KUKA KRL program: MyProgram_026().src

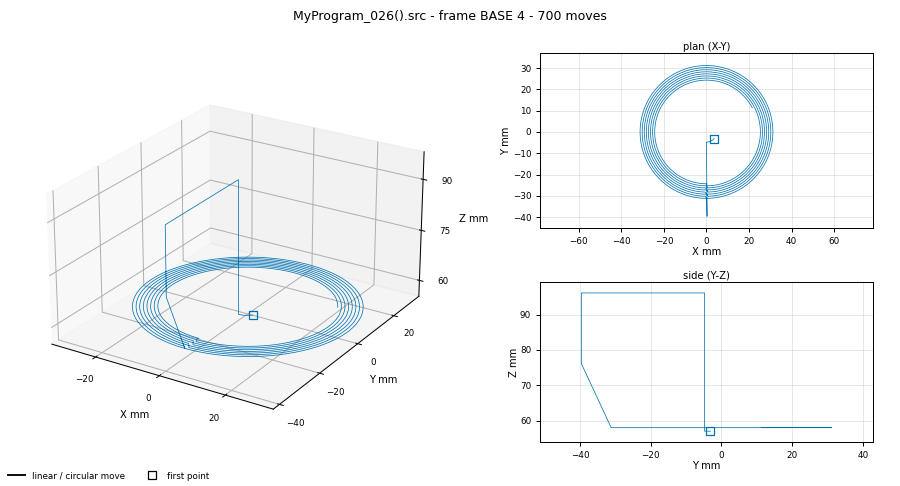
[picture p0: tool path of MyProgram_026().src in frame BASE 4, 700 of 700 moves have a stored position in this frame; points joined in program order, loops and branches not executed]
&ACCESS RVP
&REL 1
&PARAM TEMPLATE = C:\KRC\Roboter\Template\vorgabe
&PARAM EDITMASK = *
DEF MyProgram_026()
; ---- Setting reference (Base) ----
$BASE = BASE_DATA[4]

; --------------------------
; ---- Setting tool (TCP) ----
$TOOL = TOOL_DATA[3]
; --------------------------

$VEL.CP = VEL_APROX_PRINT
Startdeposition()
$VEL.CP = VEL_PRINT
LIN {X 3.5971,Y -3.1129,Z 57,A -2.6409,B 0,C 0,E1 0.1598,E2 -629.9281} C_DIS
LIN {X 2.9999,Y -3.6921,Z 57,A -2.6876,B 0,C 0,E1 0.1598,E2 -629.9281} C_DIS
LIN {X 2.3555,Y -4.1313,Z 57,A -2.7301,B 0,C 0,E1 0.1598,E2 -629.9281} C_DIS
LIN {X 1.6977,Y -4.4434,Z 57,A -2.7676,B 0,C 0,E1 0.1598,E2 -629.9281} C_DIS
LIN {X 0.8464,Y -4.6808,Z 57,A -2.809,B 0,C 0,E1 0.1598,E2 -629.9281} C_DIS
LIN {X -0.0081,Y -4.7574,Z 57,A -2.8436,B 0,C 0,E1 0.1598,E2 -629.9282} C_DIS
Enddeposition()
LIN {X -0.0081,Y -4.7574,Z 62,A -2.8335,B 0,C 0,E1 0.1598,E2 -629.928} C_DIS
LIN {X -0.0081,Y -4.7573,Z 77,A -2.8076,B 0,C 0,E1 0.1598,E2 -629.9269} C_DIS
LIN {X -0.0081,Y -4.7573,Z 96.1262,A -2.7825,B 0,C 0,E1 0.1598,E2 -629.9267} C_DIS
LIN {X 0.2603,Y -39.6445,Z 96.1262,A -95.8861,B 24.839,C -2.9274,E1 25.0032,E2 -541.4173} C_DIS
LIN {X 0.2603,Y -39.6445,Z 76.1262,A -95.5567,B 24.8539,C -2.789,E1 25.0032,E2 -541.4173} C_DIS
LIN {X 0.1436,Y -33.3063,Z 62.5315,A -95.5942,B 24.8522,C -2.8048,E1 25.0032,E2 -541.4173} C_DIS
LIN {X 0.1047,Y -31.1935,Z 58,A -95.6082,B 24.8516,C -2.8106,E1 25.0032,E2 -541.4173} C_DIS
Startdeposition()
$VEL.CP = VEL_PRINT
LIN {X 2.2949,Y -31.1109,Z 58,A -91.3981,B 24.8512,C -2.8143,E1 25.015,E2 -545.6344} C_DIS
LIN {X 4.5773,Y -30.8578,Z 58,A -87.1855,B 24.8509,C -2.8169,E1 25.0267,E2 -549.8498} C_DIS
LIN {X 6.835,Y -30.4375,Z 58,A -82.975,B 24.8506,C -2.8204,E1 25.0382,E2 -554.0634} C_DIS
LIN {X 9.0556,Y -29.8522,Z 58,A -78.7668,B 24.8501,C -2.8248,E1 25.0495,E2 -558.275} C_DIS
LIN {X 11.2271,Y -29.1051,Z 58,A -74.5606,B 24.8495,C -2.83,E1 25.0606,E2 -562.485} C_DIS
LIN {X 13.3378,Y -28.2004,Z 58,A -70.3565,B 24.8489,C -2.8362,E1 25.0713,E2 -566.6932} C_DIS
LIN {X 15.3762,Y -27.1428,Z 58,A -66.1541,B 24.8481,C -2.8431,E1 25.0816,E2 -570.8999} C_DIS
LIN {X 17.3313,Y -25.9381,Z 58,A -61.9537,B 24.8473,C -2.8508,E1 25.0915,E2 -575.1049} C_DIS
LIN {X 19.1924,Y -24.5928,Z 58,A -57.755,B 24.8464,C -2.8592,E1 25.1008,E2 -579.3084} C_DIS
LIN {X 20.9496,Y -23.1143,Z 58,A -53.558,B 24.8454,C -2.8683,E1 25.1097,E2 -583.5105} C_DIS
LIN {X 22.5932,Y -21.5105,Z 58,A -49.3625,B 24.8444,C -2.8781,E1 25.1179,E2 -587.7112} C_DIS
LIN {X 24.1144,Y -19.7902,Z 58,A -45.1683,B 24.8432,C -2.8884,E1 25.1255,E2 -591.9108} C_DIS
LIN {X 25.5049,Y -17.9626,Z 58,A -40.9754,B 24.8421,C -2.8993,E1 25.1324,E2 -596.1092} C_DIS
LIN {X 26.7572,Y -16.0377,Z 58,A -36.7836,B 24.8408,C -2.9106,E1 25.1386,E2 -600.3066} C_DIS
LIN {X 27.8645,Y -14.0258,Z 58,A -32.5927,B 24.8395,C -2.9223,E1 25.1441,E2 -604.5031} C_DIS
LIN {X 28.8208,Y -11.938,Z 58,A -28.4027,B 24.8382,C -2.9344,E1 25.1488,E2 -608.6988} C_DIS
LIN {X 29.621,Y -9.7854,Z 58,A -24.2134,B 24.8368,C -2.9467,E1 25.1527,E2 -612.8938} C_DIS
LIN {X 30.2606,Y -7.5799,Z 58,A -20.0245,B 24.8354,C -2.9593,E1 25.1557,E2 -617.0884} C_DIS
LIN {X 30.7362,Y -5.3332,Z 58,A -15.836,B 24.834,C -2.972,E1 25.1579,E2 -621.2824} C_DIS
LIN {X 31.0452,Y -3.0577,Z 58,A -11.6476,B 24.8326,C -2.9848,E1 25.1593,E2 -625.4764} C_DIS
LIN {X 31.1861,Y -0.7656,Z 58,A -8.1402,B 24.8322,C -2.9882,E1 25.1598,E2 -628.9711} C_DIS
LIN {X 31.1915,Y 0.4681,Z 58,A -5.3067,B 24.8305,C -3.0031,E1 25.1597,E2 -631.8229} C_DIS
LIN {X 31.0804,Y 2.6765,Z 58,A -1.1766,B 24.829,C -3.0166,E1 25.1589,E2 -635.9605} C_DIS
LIN {X 30.7993,Y 4.9557,Z 58,A 3.0123,B 24.8275,C -3.0291,E1 25.1573,E2 -640.1544} C_DIS
LIN {X 30.3513,Y 7.208,Z 58,A 7.2019,B 24.8261,C -3.0414,E1 25.1548,E2 -644.3487} C_DIS
LIN {X 29.7388,Y 9.4212,Z 58,A 11.392,B 24.8247,C -3.0534,E1 25.1514,E2 -648.5433} C_DIS
LIN {X 28.9652,Y 11.5834,Z 58,A 15.583,B 24.8234,C -3.065,E1 25.1473,E2 -652.7386} C_DIS
LIN {X 28.0346,Y 13.6828,Z 58,A 19.7751,B 24.8221,C -3.0763,E1 25.1423,E2 -656.9345} C_DIS
LIN {X 26.952,Y 15.7081,Z 58,A 23.9682,B 24.8208,C -3.087,E1 25.1366,E2 -661.1313} C_DIS
LIN {X 25.7234,Y 17.6483,Z 58,A 28.1627,B 24.8197,C -3.0972,E1 25.1301,E2 -665.3291} C_DIS
LIN {X 24.3555,Y 19.4928,Z 58,A 32.3584,B 24.8185,C -3.1068,E1 25.123,E2 -669.5278} C_DIS
LIN {X 22.8555,Y 21.2317,Z 58,A 36.5559,B 24.8175,C -3.1158,E1 25.1152,E2 -673.7278} C_DIS
LIN {X 21.2317,Y 22.8555,Z 58,A 40.7549,B 24.8165,C -3.1241,E1 25.1067,E2 -677.929} C_DIS
LIN {X 19.4928,Y 24.3555,Z 58,A 44.9555,B 24.8156,C -3.1316,E1 25.0977,E2 -682.1315} C_DIS
LIN {X 17.6483,Y 25.7234,Z 58,A 49.1582,B 24.8148,C -3.1384,E1 25.0881,E2 -686.3356} C_DIS
LIN {X 15.7081,Y 26.952,Z 58,A 53.3628,B 24.8141,C -3.1444,E1 25.0781,E2 -690.5412} C_DIS
LIN {X 13.6828,Y 28.0346,Z 58,A 57.5693,B 24.8135,C -3.1495,E1 25.0676,E2 -694.7483} C_DIS
LIN {X 11.5834,Y 28.9652,Z 58,A 61.7781,B 24.813,C -3.1537,E1 25.0568,E2 -698.9572} C_DIS
LIN {X 9.4212,Y 29.7388,Z 58,A 65.9888,B 24.8126,C -3.157,E1 25.0457,E2 -703.1677} C_DIS
LIN {X 7.208,Y 30.3513,Z 58,A 70.2017,B 24.8123,C -3.1595,E1 25.0343,E2 -707.38} C_DIS
LIN {X 4.9557,Y 30.7993,Z 58,A 74.4171,B 24.8121,C -3.161,E1 25.0227,E2 -711.5942} C_DIS
LIN {X 2.6765,Y 31.0804,Z 58,A 78.6345,B 24.8121,C -3.1615,E1 25.011,E2 -715.8102} C_DIS
LIN {X 0.3828,Y 31.1931,Z 58,A 82.8541,B 24.8121,C -3.1611,E1 24.9992,E2 -720.028} C_DIS
LIN {X -1.9129,Y 31.1367,Z 58,A 87.0743,B 24.8123,C -3.1597,E1 24.9875,E2 -724.2458} C_DIS
LIN {X -4.1983,Y 30.9117,Z 58,A 91.3003,B 24.8125,C -3.1575,E1 24.9757,E2 -728.4692} C_DIS
LIN {X -6.4609,Y 30.5191,Z 58,A 95.5267,B 24.8129,C -3.1543,E1 24.9642,E2 -732.6926} C_DIS
LIN {X -8.6885,Y 29.9611,Z 58,A 99.7553,B 24.8134,C -3.1501,E1 24.9528,E2 -736.9178} C_DIS
LIN {X -10.8691,Y 29.2407,Z 58,A 103.9859,B 24.814,C -3.1451,E1 24.9416,E2 -741.1448} C_DIS
LIN {X -12.9907,Y 28.3619,Z 58,A 108.2187,B 24.8147,C -3.1393,E1 24.9308,E2 -745.3735} C_DIS
LIN {X -15.0419,Y 27.3294,Z 58,A 112.4534,B 24.8155,C -3.1326,E1 24.9204,E2 -749.6039} C_DIS
LIN {X -17.0117,Y 26.1488,Z 58,A 116.6901,B 24.8164,C -3.1251,E1 24.9104,E2 -753.836} C_DIS
LIN {X -18.8892,Y 24.8265,Z 58,A 120.9285,B 24.8174,C -3.1168,E1 24.9008,E2 -758.0696} C_DIS
LIN {X -20.6644,Y 23.3697,Z 58,A 125.1687,B 24.8184,C -3.1078,E1 24.8918,E2 -762.3048} C_DIS
LIN {X -22.3275,Y 21.7862,Z 58,A 129.4103,B 24.8195,C -3.0982,E1 24.8834,E2 -766.5412} C_DIS
LIN {X -23.8697,Y 20.0846,Z 58,A 133.6535,B 24.8207,C -3.0879,E1 24.8756,E2 -770.779} C_DIS
LIN {X -25.2826,Y 18.2742,Z 58,A 137.8979,B 24.822,C -3.0771,E1 24.8685,E2 -775.018} C_DIS
LIN {X -26.5584,Y 16.3648,Z 58,A 142.1437,B 24.8233,C -3.0658,E1 24.8621,E2 -779.2582} C_DIS
LIN {X -27.6903,Y 14.3667,Z 58,A 146.3904,B 24.8247,C -3.0541,E1 24.8565,E2 -783.4992} C_DIS
LIN {X -28.6722,Y 12.2908,Z 58,A 150.638,B 24.8261,C -3.042,E1 24.8516,E2 -787.7411} C_DIS
LIN {X -29.4987,Y 10.1482,Z 58,A 154.8864,B 24.8275,C -3.0296,E1 24.8476,E2 -791.9838} C_DIS
LIN {X -30.1653,Y 7.9506,Z 58,A 159.1351,B 24.8289,C -3.0169,E1 24.8443,E2 -796.2268} C_DIS
LIN {X -30.6684,Y 5.71,Z 58,A 163.3845,B 24.8304,C -3.0041,E1 24.842,E2 -800.4706} C_DIS
LIN {X -31.0054,Y 3.4384,Z 58,A 167.634,B 24.8318,C -2.9912,E1 24.8405,E2 -804.7145} C_DIS
LIN {X -31.1743,Y 1.1482,Z 58,A 171.597,B 24.8335,C -2.9761,E1 24.8398,E2 -808.6653} C_DIS
LIN {X -31.1861,Y -0.7656,Z 58,A 175.4249,B 24.8345,C -2.9675,E1 24.8399,E2 -812.4955} C_DIS
LIN {X -31.0452,Y -3.0577,Z 58,A 179.674,B 24.8359,C -2.9547,E1 24.8409,E2 -816.7395} C_DIS
LIN {X -30.7362,Y -5.3332,Z 58,A -176.0771,B 24.8373,C -2.942,E1 24.8427,E2 -820.9834} C_DIS
LIN {X -30.2606,Y -7.5799,Z 58,A -171.8289,B 24.8387,C -2.9296,E1 24.8454,E2 -825.2269} C_DIS
LIN {X -29.621,Y -9.7854,Z 58,A -167.5814,B 24.84,C -2.9176,E1 24.8489,E2 -829.4699} C_DIS
LIN {X -28.8208,Y -11.938,Z 58,A -163.3348,B 24.8413,C -2.9059,E1 24.8532,E2 -833.7123} C_DIS
LIN {X -27.8645,Y -14.0258,Z 58,A -159.0893,B 24.8426,C -2.8946,E1 24.8583,E2 -837.954} C_DIS
LIN {X -26.7572,Y -16.0377,Z 58,A -154.845,B 24.8437,C -2.8839,E1 24.8642,E2 -842.1947} C_DIS
LIN {X -25.5049,Y -17.9626,Z 58,A -150.602,B 24.8448,C -2.8737,E1 24.8709,E2 -846.4344} C_DIS
LIN {X -24.1144,Y -19.7902,Z 58,A -146.3605,B 24.8459,C -2.8641,E1 24.8782,E2 -850.673} C_DIS
LIN {X -22.5932,Y -21.5105,Z 58,A -142.1207,B 24.8468,C -2.8553,E1 24.8862,E2 -854.9103} C_DIS
LIN {X -20.9496,Y -23.1143,Z 58,A -137.8825,B 24.8477,C -2.8471,E1 24.8948,E2 -859.1464} C_DIS
LIN {X -19.1924,Y -24.5928,Z 58,A -133.6461,B 24.8485,C -2.8397,E1 24.904,E2 -863.381} C_DIS
LIN {X -17.3313,Y -25.9381,Z 58,A -129.4116,B 24.8492,C -2.8331,E1 24.9137,E2 -867.6141} C_DIS
LIN {X -15.3762,Y -27.1428,Z 58,A -125.1792,B 24.8498,C -2.8274,E1 24.9239,E2 -871.8456} C_DIS
LIN {X -13.3378,Y -28.2004,Z 58,A -120.9489,B 24.8503,C -2.8225,E1 24.9345,E2 -876.0755} C_DIS
LIN {X -11.2271,Y -29.1051,Z 58,A -116.7206,B 24.8508,C -2.8185,E1 24.9454,E2 -880.3037} C_DIS
LIN {X -9.0556,Y -29.8522,Z 58,A -112.4946,B 24.8511,C -2.8154,E1 24.9567,E2 -884.53} C_DIS
LIN {X -6.835,Y -30.4375,Z 58,A -108.2707,B 24.8513,C -2.8133,E1 24.9681,E2 -888.7546} C_DIS
LIN {X -4.5773,Y -30.8578,Z 58,A -104.0493,B 24.8514,C -2.8121,E1 24.9797,E2 -892.9773} C_DIS
LIN {X -2.2949,Y -31.1109,Z 58,A -99.8299,B 24.8514,C -2.8119,E1 24.9915,E2 -897.1982} C_DIS
LIN {X 0.1047,Y -31.1935,Z 58,A -95.6081,B 24.8516,C -2.8106,E1 25.0033,E2 -901.4173} C_DIS
Enddeposition()
LIN {X 0.1047,Y -31.1935,Z 58,A -95.6081,B 24.8516,C -2.8106,E1 25.0033,E2 -901.4173} C_DIS
Startdeposition()
$VEL.CP = VEL_PRINT
LIN {X -0.5457,Y -30.2108,Z 58,A -98.6907,B 24.8519,C -2.8079,E1 24.9946,E2 -898.3283} C_DIS
LIN {X -2.6136,Y -30.1028,Z 58,A -102.6666,B 24.8519,C -2.8074,E1 24.9835,E2 -894.3496} C_DIS
LIN {X -4.817,Y -29.8297,Z 58,A -106.8223,B 24.8518,C -2.8088,E1 24.9721,E2 -890.194} C_DIS
LIN {X -6.6677,Y -29.4712,Z 58,A -110.3863,B 24.8516,C -2.8104,E1 24.9623,E2 -886.6296} C_DIS
LIN {X -9.1107,Y -28.8099,Z 58,A -115.271,B 24.8514,C -2.8128,E1 24.9492,E2 -881.7424} C_DIS
LIN {X -11.2355,Y -28.0496,Z 58,A -119.5455,B 24.851,C -2.8166,E1 24.9381,E2 -877.4682} C_DIS
LIN {X -13.2679,Y -27.1474,Z 58,A -123.8987,B 24.8506,C -2.8202,E1 24.927,E2 -873.1125} C_DIS
LIN {X -15.1376,Y -26.1506,Z 58,A -127.6644,B 24.8498,C -2.8276,E1 24.9179,E2 -869.3537} C_DIS
LIN {X -16.7352,Y -25.1583,Z 58,A -131.3179,B 24.8493,C -2.8322,E1 24.9093,E2 -865.6995} C_DIS
LIN {X -18.2715,Y -24.0658,Z 58,A -134.908,B 24.8487,C -2.8381,E1 24.9012,E2 -862.1106} C_DIS
LIN {X -19.7968,Y -22.8273,Z 58,A -138.5955,B 24.8479,C -2.8452,E1 24.8933,E2 -858.4261} C_DIS
LIN {X -21.2071,Y -21.5232,Z 58,A -142.6762,B 24.8475,C -2.8491,E1 24.8851,E2 -854.3376} C_DIS
LIN {X -22.8019,Y -19.8259,Z 58,A -147.2693,B 24.8466,C -2.8574,E1 24.8766,E2 -849.7438} C_DIS
LIN {X -24.601,Y -17.5437,Z 58,A -152.3405,B 24.8448,C -2.8737,E1 24.8681,E2 -844.6872} C_DIS
LIN {X -25.8525,Y -15.6411,Z 58,A -156.1895,B 24.8433,C -2.888,E1 24.8623,E2 -840.853} C_DIS
LIN {X -26.6221,Y -14.2922,Z 58,A -159.6438,B 24.8429,C -2.892,E1 24.8576,E2 -837.3901} C_DIS
LIN {X -27.5197,Y -12.4764,Z 58,A -163.3944,B 24.8416,C -2.9031,E1 24.8531,E2 -833.6458} C_DIS
LIN {X -28.3033,Y -10.5797,Z 58,A -167.0641,B 24.8403,C -2.9156,E1 24.8494,E2 -829.9855} C_DIS
LIN {X -28.8908,Y -8.85,Z 58,A -171.2263,B 24.8397,C -2.9208,E1 24.8458,E2 -825.812} C_DIS
LIN {X -29.507,Y -6.506,Z 58,A -175.4387,B 24.8379,C -2.9372,E1 24.843,E2 -821.614} C_DIS
LIN {X -29.8601,Y -4.6221,Z 58,A -179.4869,B 24.837,C -2.9454,E1 24.8412,E2 -817.5615} C_DIS
LIN {X -30.0965,Y -2.6829,Z 58,A 177.5499,B 24.8351,C -2.9618,E1 24.8403,E2 -814.6198} C_DIS
LIN {X -30.1951,Y -1.1291,Z 58,A 174.0998,B 24.8345,C -2.9676,E1 24.8398,E2 -811.1628} C_DIS
LIN {X -30.2137,Y 0.3884,Z 58,A 171.1347,B 24.8335,C -2.976,E1 24.8398,E2 -808.2} C_DIS
LIN {X -30.0111,Y 3.506,Z 58,A 164.6989,B 24.8318,C -2.9911,E1 24.8414,E2 -801.7618} C_DIS
LIN {X -29.5072,Y 6.5047,Z 58,A 158.887,B 24.8299,C -3.0087,E1 24.8445,E2 -795.9576} C_DIS
LIN {X -28.8455,Y 8.9959,Z 58,A 154.669,B 24.8276,C -3.0281,E1 24.8478,E2 -791.7616} C_DIS
LIN {X -28.2324,Y 10.7669,Z 58,A 150.9243,B 24.8266,C -3.0375,E1 24.8513,E2 -788.0182} C_DIS
LIN {X -27.3464,Y 12.852,Z 58,A 146.3112,B 24.8254,C -3.0479,E1 24.8566,E2 -783.4046} C_DIS
LIN {X -25.9429,Y 15.491,Z 58,A 140.9017,B 24.8233,C -3.0656,E1 24.8639,E2 -778.0093} C_DIS
LIN {X -24.8443,Y 17.1975,Z 58,A 137.0408,B 24.8221,C -3.0759,E1 24.8699,E2 -774.1538} C_DIS
LIN {X -23.5808,Y 18.8935,Z 58,A 132.9127,B 24.821,C -3.0855,E1 24.877,E2 -770.0289} C_DIS
LIN {X -22.0567,Y 20.6518,Z 58,A 128.4632,B 24.8198,C -3.096,E1 24.8853,E2 -765.5849} C_DIS
LIN {X -20.8476,Y 21.8722,Z 58,A 125.6303,B 24.8185,C -3.1067,E1 24.8909,E2 -762.7657} C_DIS
LIN {X -19.1986,Y 23.3329,Z 58,A 121.0011,B 24.8179,C -3.1124,E1 24.9007,E2 -758.132} C_DIS
LIN {X -17.428,Y 24.6835,Z 58,A 116.7503,B 24.8169,C -3.1206,E1 24.9102,E2 -753.8859} C_DIS
LIN {X -15.6312,Y 25.8585,Z 58,A 112.7849,B 24.8159,C -3.1289,E1 24.9196,E2 -749.9277} C_DIS
LIN {X -13.8263,Y 26.8669,Z 58,A 109.5725,B 24.8145,C -3.1412,E1 24.9274,E2 -746.7355} C_DIS
LIN {X -12.1506,Y 27.6651,Z 58,A 104.5873,B 24.8153,C -3.1342,E1 24.9401,E2 -741.7214} C_DIS
LIN {X -9.6521,Y 28.6326,Z 58,A 100.3116,B 24.8137,C -3.1474,E1 24.9513,E2 -737.4684} C_DIS
LIN {X -7.4806,Y 29.2751,Z 58,A 95.3533,B 24.8139,C -3.1459,E1 24.9647,E2 -732.499} C_DIS
LIN {X -4.8516,Y 29.824,Z 58,A 90.8217,B 24.8128,C -3.1548,E1 24.9771,E2 -727.9839} C_DIS
LIN {X -2.895,Y 30.0769,Z 58,A 87.058,B 24.8126,C -3.1566,E1 24.9875,E2 -724.2221} C_DIS
LIN {X -0.8345,Y 30.2043,Z 58,A 83.1681,B 24.8124,C -3.1582,E1 24.9984,E2 -720.3349} C_DIS
LIN {X 1.0968,Y 30.1963,Z 58,A 79.3527,B 24.8126,C -3.1572,E1 25.009,E2 -716.5178} C_DIS
LIN {X 2.9201,Y 30.0746,Z 58,A 76.1368,B 24.8123,C -3.1594,E1 25.0179,E2 -713.3089} C_DIS
LIN {X 4.4982,Y 29.8786,Z 58,A 73.3207,B 24.8121,C -3.1607,E1 25.0257,E2 -710.4984} C_DIS
LIN {X 6.1892,Y 29.5752,Z 58,A 69.76,B 24.8127,C -3.1563,E1 25.0355,E2 -706.9313} C_DIS
LIN {X 8.1432,Y 29.0979,Z 58,A 65.9758,B 24.8129,C -3.1543,E1 25.0457,E2 -703.1483} C_DIS
LIN {X 10.3307,Y 28.3948,Z 58,A 61.382,B 24.8136,C -3.1482,E1 25.0579,E2 -698.549} C_DIS
LIN {X 12.0292,Y 27.718,Z 58,A 57.7365,B 24.8143,C -3.1427,E1 25.0673,E2 -694.899} C_DIS
LIN {X 14.7973,Y 26.3445,Z 58,A 52.3919,B 24.8145,C -3.141,E1 25.0805,E2 -689.5652} C_DIS
LIN {X 16.4389,Y 25.3529,Z 58,A 48.6582,B 24.8153,C -3.1345,E1 25.0893,E2 -685.828} C_DIS
LIN {X 17.6927,Y 24.4946,Z 58,A 46.1986,B 24.8153,C -3.1346,E1 25.0949,E2 -683.3773} C_DIS
LIN {X 19.3952,Y 23.1695,Z 58,A 41.6642,B 24.8167,C -3.1221,E1 25.1048,E2 -678.8302} C_DIS
LIN {X 20.9276,Y 21.7951,Z 58,A 37.7631,B 24.8176,C -3.1145,E1 25.1128,E2 -674.9267} C_DIS
LIN {X 22.3953,Y 20.2847,Z 58,A 33.7242,B 24.8187,C -3.1054,E1 25.1205,E2 -670.8838} C_DIS
LIN {X 23.411,Y 19.103,Z 58,A 30.8393,B 24.8194,C -3.0995,E1 25.1257,E2 -667.9983} C_DIS
LIN {X 24.5993,Y 17.5459,Z 58,A 27.1691,B 24.8204,C -3.0912,E1 25.1318,E2 -664.326} C_DIS
LIN {X 25.7265,Y 15.8484,Z 58,A 23.3683,B 24.8214,C -3.0822,E1 25.1375,E2 -660.5231} C_DIS
LIN {X 26.864,Y 13.832,Z 58,A 19.7293,B 24.8216,C -3.0801,E1 25.1424,E2 -656.8981} C_DIS
LIN {X 27.5705,Y 12.3637,Z 58,A 15.7043,B 24.824,C -3.0598,E1 25.1472,E2 -652.8466} C_DIS
LIN {X 28.4448,Y 10.1938,Z 58,A 11.413,B 24.8252,C -3.049,E1 25.1514,E2 -648.5537} C_DIS
LIN {X 29.1291,Y 8.0317,Z 58,A 7.1909,B 24.8266,C -3.0374,E1 25.1548,E2 -644.3282} C_DIS
LIN {X 29.6149,Y 5.9961,Z 58,A 3.4136,B 24.8277,C -3.0279,E1 25.1571,E2 -640.5506} C_DIS
LIN {X 29.8676,Y 4.5736,Z 58,A 0.5902,B 24.8287,C -3.0185,E1 25.1583,E2 -637.7214} C_DIS
LIN {X 30.1344,Y 2.2217,Z 58,A -3.8278,B 24.8302,C -3.0056,E1 25.1595,E2 -633.2989} C_DIS
LIN {X 30.217,Y 0.2137,Z 58,A -7.7625,B 24.8317,C -2.992,E1 25.1598,E2 -629.3555} C_DIS
LIN {X 30.1601,Y -1.8398,Z 58,A -11.6005,B 24.833,C -2.9806,E1 25.1593,E2 -625.5133} C_DIS
LIN {X 29.9414,Y -4.0661,Z 58,A -15.82,B 24.8345,C -2.9677,E1 25.1579,E2 -621.2881} C_DIS
LIN {X 29.5704,Y -6.211,Z 58,A -19.9239,B 24.8359,C -2.9552,E1 25.1558,E2 -617.1786} C_DIS
LIN {X 28.9354,Y -8.7031,Z 58,A -24.6878,B 24.8374,C -2.9417,E1 25.1523,E2 -612.41} C_DIS
LIN {X 28.4876,Y -10.0724,Z 58,A -27.3182,B 24.8382,C -2.9347,E1 25.1499,E2 -609.7781} C_DIS
LIN {X 27.8924,Y -11.6196,Z 58,A -30.5996,B 24.8394,C -2.9236,E1 25.1464,E2 -606.4884} C_DIS
LIN {X 26.9378,Y -13.6875,Z 58,A -34.8414,B 24.8407,C -2.912,E1 25.1413,E2 -602.2419} C_DIS
LIN {X 25.9819,Y -15.425,Z 58,A -38.355,B 24.8415,C -2.9045,E1 25.1364,E2 -598.729} C_DIS
LIN {X 24.9527,Y -17.0402,Z 58,A -42.4302,B 24.8432,C -2.889,E1 25.1301,E2 -594.6372} C_DIS
LIN {X 23.6005,Y -18.8688,Z 58,A -46.5529,B 24.8441,C -2.8801,E1 25.1231,E2 -590.513} C_DIS
LIN {X 22.5055,Y -20.1616,Z 58,A -50.3292,B 24.8458,C -2.8652,E1 25.116,E2 -586.7182} C_DIS
LIN {X 20.552,Y -22.1502,Z 58,A -54.8613,B 24.8461,C -2.8621,E1 25.107,E2 -582.1975} C_DIS
LIN {X 18.814,Y -23.6439,Z 58,A -59.3971,B 24.8474,C -2.8503,E1 25.0972,E2 -577.6514} C_DIS
LIN {X 16.9476,Y -25.0154,Z 58,A -63.4494,B 24.8479,C -2.8457,E1 25.088,E2 -573.602} C_DIS
LIN {X 15.2508,Y -26.0849,Z 58,A -67.3504,B 24.8487,C -2.8376,E1 25.0787,E2 -569.6941} C_DIS
LIN {X 13.6015,Y -26.9818,Z 58,A -70.5396,B 24.8489,C -2.836,E1 25.0708,E2 -566.5102} C_DIS
LIN {X 12.2067,Y -27.6406,Z 58,A -74.8667,B 24.8511,C -2.8157,E1 25.0597,E2 -562.1455} C_DIS
LIN {X 8.0206,Y -29.132,Z 58,A -81.8375,B 24.8504,C -2.8219,E1 25.0413,E2 -555.2027} C_DIS
LIN {X 5.5141,Y -29.7077,Z 58,A -87.7303,B 24.852,C -2.8066,E1 25.0251,E2 -549.2812} C_DIS
LIN {X 2.6715,Y -30.0976,Z 58,A -92.811,B 24.852,C -2.8073,E1 25.011,E2 -544.2057} C_DIS
LIN {X 0.6893,Y -30.2073,Z 58,A -96.4907,B 24.852,C -2.8069,E1 25.0008,E2 -540.5259} C_DIS
LIN {X 0.6893,Y -30.2073,Z 58,A -96.4907,B 24.852,C -2.8069,E1 25.0008,E2 -540.5259} C_DIS
Enddeposition()
LIN {X 0.0903,Y -29.2216,Z 58,A -96.0606,B 24.8485,C -2.8398,E1 25.0022,E2 -541.0343} C_DIS
Startdeposition()
$VEL.CP = VEL_PRINT
LIN {X 2.9841,Y -29.0837,Z 58,A -90.6247,B 24.8485,C -2.8394,E1 25.0173,E2 -546.467} C_DIS
LIN {X 4.2179,Y -28.9307,Z 58,A -87.8707,B 24.848,C -2.8443,E1 25.025,E2 -549.2304} C_DIS
LIN {X 5.7719,Y -28.6613,Z 58,A -84.2426,B 24.8471,C -2.8525,E1 25.035,E2 -552.8739} C_DIS
LIN {X 7.6559,Y -28.2164,Z 58,A -80.4789,B 24.8468,C -2.856,E1 25.0452,E2 -556.6401} C_DIS
LIN {X 9.6009,Y -27.6152,Z 58,A -76.4651,B 24.8462,C -2.861,E1 25.0558,E2 -560.6582} C_DIS
LIN {X 11.7718,Y -26.7621,Z 58,A -72.1374,B 24.8458,C -2.8647,E1 25.067,E2 -564.9846} C_DIS
LIN {X 13.7475,Y -25.8031,Z 58,A -67.6863,B 24.8449,C -2.8733,E1 25.0781,E2 -569.4439} C_DIS
LIN {X 15.4832,Y -24.8001,Z 58,A -63.8818,B 24.8443,C -2.8789,E1 25.0872,E2 -573.25} C_DIS
LIN {X 17.236,Y -23.6156,Z 58,A -59.9967,B 24.8437,C -2.884,E1 25.0961,E2 -577.1338} C_DIS
LIN {X 18.7,Y -22.4741,Z 58,A -55.9309,B 24.8423,C -2.897,E1 25.1049,E2 -581.2149} C_DIS
LIN {X 19.9329,Y -21.3884,Z 58,A -52.9556,B 24.8418,C -2.9013,E1 25.1111,E2 -584.1885} C_DIS
LIN {X 21.4288,Y -19.89,Z 58,A -49.0802,B 24.8411,C -2.9078,E1 25.1186,E2 -588.0628} C_DIS
LIN {X 22.5343,Y -18.6276,Z 58,A -46.1131,B 24.8406,C -2.9121,E1 25.124,E2 -591.0265} C_DIS
LIN {X 23.4448,Y -17.4679,Z 58,A -42.6102,B 24.839,C -2.9274,E1 25.13,E2 -594.549} C_DIS
LIN {X 24.478,Y -15.988,Z 58,A -39.0736,B 24.8379,C -2.937,E1 25.1355,E2 -598.0908} C_DIS
LIN {X 25.7366,Y -13.8706,Z 58,A -34.3702,B 24.8366,C -2.949,E1 25.142,E2 -602.7983} C_DIS
LIN {X 26.4585,Y -12.4392,Z 58,A -31.5848,B 24.8361,C -2.9536,E1 25.1454,E2 -605.5796} C_DIS
LIN {X 27.1196,Y -10.923,Z 58,A -27.9375,B 24.8344,C -2.9684,E1 25.1493,E2 -609.242} C_DIS
LIN {X 27.6966,Y -9.3633,Z 58,A -24.7331,B 24.8334,C -2.9775,E1 25.1523,E2 -612.45} C_DIS
LIN {X 28.2872,Y -7.3906,Z 58,A -21.0515,B 24.8325,C -2.9853,E1 25.1551,E2 -616.1288} C_DIS
LIN {X 28.607,Y -6.0368,Z 58,A -18.2439,B 24.8314,C -2.9948,E1 25.1568,E2 -618.9426} C_DIS
LIN {X 28.8647,Y -4.648,Z 58,A -15.5364,B 24.8305,C -3.0026,E1 25.1581,E2 -621.6528} C_DIS
LIN {X 29.0991,Y -2.8354,Z 58,A -11.7261,B 24.8289,C -3.0168,E1 25.1593,E2 -625.4742} C_DIS
LIN {X 29.2277,Y -0.7351,Z 58,A -7.7496,B 24.8277,C -3.0278,E1 25.1598,E2 -629.453} C_DIS
LIN {X 29.2047,Y 1.3684,Z 58,A -3.1312,B 24.8255,C -3.0471,E1 25.1594,E2 -634.0897} C_DIS
LIN {X 29.001,Y 3.7038,Z 58,A 0.9813,B 24.8246,C -3.055,E1 25.1581,E2 -638.1964} C_DIS
LIN {X 28.66,Y 5.7783,Z 58,A 4.711,B 24.8237,C -3.0624,E1 25.1563,E2 -641.922} C_DIS
LIN {X 28.278,Y 7.4264,Z 58,A 8.4733,B 24.8219,C -3.078,E1 25.1538,E2 -645.6996} C_DIS
LIN {X 27.6453,Y 9.5155,Z 58,A 13.3726,B 24.8195,C -3.0984,E1 25.1495,E2 -650.6194} C_DIS
LIN {X 26.8792,Y 11.5026,Z 58,A 16.87,B 24.8191,C -3.1015,E1 25.1457,E2 -654.1049} C_DIS
LIN {X 26.1324,Y 13.1102,Z 58,A 20.0015,B 24.8185,C -3.1066,E1 25.1419,E2 -657.2317} C_DIS
LIN {X 25.3083,Y 14.6381,Z 58,A 23.1856,B 24.8178,C -3.1129,E1 25.1376,E2 -660.414} C_DIS
LIN {X 24.4611,Y 16.0137,Z 58,A 26.8475,B 24.8162,C -3.127,E1 25.1321,E2 -664.091} C_DIS
LIN {X 23.4636,Y 17.4426,Z 58,A 30.2219,B 24.8152,C -3.1347,E1 25.1266,E2 -667.4674} C_DIS
LIN {X 22.2021,Y 19.0223,Z 58,A 34.4022,B 24.8139,C -3.1463,E1 25.1191,E2 -671.656} C_DIS
LIN {X 20.2402,Y 21.0978,Z 58,A 39.3304,B 24.8134,C -3.15,E1 25.1095,E2 -676.5719} C_DIS
LIN {X 18.4609,Y 22.671,Z 58,A 44.7663,B 24.8113,C -3.1679,E1 25.0979,E2 -682.0291} C_DIS
LIN {X 16.4708,Y 24.1557,Z 58,A 48.7743,B 24.8115,C -3.1661,E1 25.0889,E2 -686.0188} C_DIS
LIN {X 15.057,Y 25.0616,Z 58,A 52.5048,B 24.8103,C -3.1759,E1 25.08,E2 -689.7607} C_DIS
LIN {X 12.8183,Y 26.2765,Z 58,A 57.4825,B 24.8096,C -3.1821,E1 25.0677,E2 -694.7392} C_DIS
LIN {X 11.2938,Y 26.9672,Z 58,A 60.3474,B 24.8097,C -3.1811,E1 25.0604,E2 -697.5947} C_DIS
LIN {X 9.9654,Y 27.4858,Z 58,A 63.2885,B 24.8092,C -3.1852,E1 25.0527,E2 -700.5394} C_DIS
LIN {X 8.1782,Y 28.0698,Z 58,A 66.9458,B 24.8089,C -3.1876,E1 25.0429,E2 -704.1958} C_DIS
LIN {X 6.3939,Y 28.5293,Z 58,A 71.6057,B 24.8074,C -3.2004,E1 25.0302,E2 -708.8796} C_DIS
LIN {X 3.1402,Y 29.0675,Z 58,A 76.8496,B 24.8087,C -3.1897,E1 25.0158,E2 -714.0934} C_DIS
LIN {X 1.8901,Y 29.1755,Z 58,A 80.2187,B 24.8076,C -3.1987,E1 25.0063,E2 -717.4823} C_DIS
LIN {X -1.4179,Y 29.2026,Z 58,A 85.5477,B 24.8091,C -3.1862,E1 24.9915,E2 -722.7816} C_DIS
LIN {X -2.6099,Y 29.1199,Z 58,A 89.1479,B 24.8078,C -3.1968,E1 24.9814,E2 -726.409} C_DIS
LIN {X -5.548,Y 28.7053,Z 58,A 94.3405,B 24.809,C -3.1871,E1 24.9672,E2 -731.5832} C_DIS
LIN {X -7.6313,Y 28.223,Z 58,A 98.8076,B 24.8092,C -3.1856,E1 24.9551,E2 -736.053} C_DIS
LIN {X -9.3929,Y 27.6866,Z 58,A 102.151,B 24.8099,C -3.1791,E1 24.9462,E2 -739.3872} C_DIS
LIN {X -12.1362,Y 26.599,Z 58,A 108.7196,B 24.8101,C -3.1777,E1 24.9293,E2 -745.9675} C_DIS
LIN {X -14.1754,Y 25.5703,Z 58,A 113.3874,B 24.8108,C -3.1718,E1 24.9179,E2 -750.6345} C_DIS
LIN {X -17.5086,Y 23.4143,Z 58,A 119.4587,B 24.8142,C -3.1435,E1 24.9039,E2 -756.6584} C_DIS
LIN {X -18.6997,Y 22.4744,Z 58,A 123.5779,B 24.8139,C -3.146,E1 24.895,E2 -760.799} C_DIS
LIN {X -20.5269,Y 20.8187,Z 58,A 128.1212,B 24.8155,C -3.1328,E1 24.8858,E2 -765.3293} C_DIS
LIN {X -22.8174,Y 18.2799,Z 58,A 136.0694,B 24.8164,C -3.1252,E1 24.8713,E2 -773.2956} C_DIS
LIN {X -24.6357,Y 15.7433,Z 58,A 141.8127,B 24.8186,C -3.106,E1 24.8625,E2 -779.0216} C_DIS
LIN {X -26.3279,Y 12.713,Z 58,A 147.4846,B 24.8218,C -3.0788,E1 24.8551,E2 -784.6584} C_DIS
LIN {X -26.8596,Y 11.548,Z 58,A 150.2427,B 24.8225,C -3.0731,E1 24.852,E2 -787.4181} C_DIS
LIN {X -27.5231,Y 9.8631,Z 58,A 153.8884,B 24.8236,C -3.0631,E1 24.8484,E2 -791.0605} C_DIS
LIN {X -28.1658,Y 7.8389,Z 58,A 158.0814,B 24.8251,C -3.0507,E1 24.845,E2 -795.2479} C_DIS
LIN {X -28.6179,Y 5.9833,Z 58,A 161.9339,B 24.8263,C -3.0399,E1 24.8426,E2 -799.0971} C_DIS
LIN {X -28.984,Y 3.8347,Z 58,A 166.5756,B 24.8275,C -3.0291,E1 24.8407,E2 -803.7406} C_DIS
LIN {X -29.1636,Y 2.0625,Z 58,A 169.7663,B 24.829,C -3.0162,E1 24.84,E2 -806.9195} C_DIS
LIN {X -29.2367,Y 0.034,Z 58,A 173.9631,B 24.8303,C -3.0052,E1 24.8398,E2 -811.1154} C_DIS
LIN {X -29.1417,Y -2.3528,Z 58,A 178.2848,B 24.8322,C -2.9883,E1 24.8405,E2 -815.4226} C_DIS
LIN {X -28.8334,Y -4.8382,Z 58,A -175.7906,B 24.8331,C -2.9802,E1 24.8429,E2 -821.3631} C_DIS
LIN {X -28.1999,Y -7.7166,Z 58,A -171.1421,B 24.8359,C -2.9552,E1 24.8459,E2 -825.979} C_DIS
LIN {X -27.8108,Y -9.0186,Z 58,A -168.259,B 24.8366,C -2.949,E1 24.8483,E2 -828.8637} C_DIS
LIN {X -27.3689,Y -10.2821,Z 58,A -165.7718,B 24.8375,C -2.9406,E1 24.8507,E2 -831.3448} C_DIS
LIN {X -26.7671,Y -11.7601,Z 58,A -162.2213,B 24.8381,C -2.9348,E1 24.8546,E2 -834.9013} C_DIS
LIN {X -25.8501,Y -13.6584,Z 58,A -157.6261,B 24.839,C -2.9271,E1 24.8604,E2 -839.5025} C_DIS
LIN {X -24.5268,Y -15.9132,Z 58,A -152.8732,B 24.8407,C -2.9114,E1 24.8674,E2 -844.2421} C_DIS
LIN {X -23.4965,Y -17.3985,Z 58,A -149.6203,B 24.8419,C -2.9007,E1 24.8726,E2 -847.4853} C_DIS
LIN {X -22.5946,Y -18.5543,Z 58,A -146.603,B 24.8425,C -2.8952,E1 24.8779,E2 -850.5036} C_DIS
LIN {X -21.3809,Y -19.941,Z 58,A -142.7519,B 24.8432,C -2.8892,E1 24.8851,E2 -854.3575} C_DIS
LIN {X -20.0076,Y -21.3183,Z 58,A -139.4764,B 24.8444,C -2.8773,E1 24.8917,E2 -857.6183} C_DIS
LIN {X -19.1442,Y -22.0972,Z 58,A -136.6959,B 24.8444,C -2.877,E1 24.8975,E2 -860.409} C_DIS
LIN {X -17.5445,Y -23.3873,Z 58,A -132.7798,B 24.8453,C -2.8691,E1 24.9061,E2 -864.3205} C_DIS
LIN {X -15.9811,Y -24.4826,Z 58,A -128.8654,B 24.8458,C -2.8647,E1 24.9152,E2 -868.2375} C_DIS
LIN {X -14.109,Y -25.6069,Z 58,A -125.0227,B 24.8469,C -2.8551,E1 24.9245,E2 -872.0687} C_DIS
LIN {X -12.8814,Y -26.2461,Z 58,A -122.1321,B 24.847,C -2.8534,E1 24.9317,E2 -874.963} C_DIS
LIN {X -11.2431,Y -26.9886,Z 58,A -118.3449,B 24.8472,C -2.852,E1 24.9414,E2 -878.7559} C_DIS
LIN {X -9.2986,Y -27.7185,Z 58,A -113.7086,B 24.847,C -2.8539,E1 24.9536,E2 -883.4057} C_DIS
LIN {X -6.5795,Y -28.4864,Z 58,A -108.9226,B 24.8481,C -2.8437,E1 24.9665,E2 -888.1745} C_DIS
LIN {X -4.7345,Y -28.8508,Z 58,A -105.6843,B 24.8487,C -2.8382,E1 24.9754,E2 -891.403} C_DIS
LIN {X -3.5496,Y -29.0206,Z 58,A -102.7499,B 24.8481,C -2.8435,E1 24.9836,E2 -894.3521} C_DIS
LIN {X -1.6541,Y -29.1897,Z 58,A -98.9798,B 24.8481,C -2.8439,E1 24.9941,E2 -898.1246} C_DIS
LIN {X 0.0903,Y -29.2216,Z 58,A -96.0604,B 24.8485,C -2.8397,E1 25.0022,E2 -901.0343} C_DIS
Enddeposition()
LIN {X 0.0903,Y -29.2216,Z 58,A -96.0604,B 24.8485,C -2.8397,E1 25.0022,E2 -901.0343} C_DIS
Startdeposition()
$VEL.CP = VEL_PRINT
LIN {X -0.6743,Y -28.2497,Z 58,A -98.8134,B 24.848,C -2.8444,E1 24.9945,E2 -898.2923} C_DIS
LIN {X -3.3063,Y -28.0633,Z 58,A -105.1324,B 24.8489,C -2.8358,E1 24.9769,E2 -891.9496} C_DIS
LIN {X -5.4836,Y -27.7202,Z 58,A -109.5833,B 24.8487,C -2.8375,E1 24.9647,E2 -887.4982} C_DIS
LIN {X -8.6576,Y -26.898,Z 58,A -115.5253,B 24.8476,C -2.8478,E1 24.9488,E2 -881.5712} C_DIS
LIN {X -10.8271,Y -26.101,Z 58,A -120.556,B 24.8475,C -2.8493,E1 24.9357,E2 -876.5332} C_DIS
LIN {X -12.7919,Y -25.1962,Z 58,A -124.6533,B 24.8467,C -2.8567,E1 24.9254,E2 -872.4429} C_DIS
LIN {X -14.5409,Y -24.2295,Z 58,A -128.7773,B 24.8461,C -2.8616,E1 24.9154,E2 -868.3185} C_DIS
LIN {X -16.3,Y -23.0826,Z 58,A -133.1017,B 24.8455,C -2.8678,E1 24.9054,E2 -863.9943} C_DIS
LIN {X -17.9549,Y -21.8201,Z 58,A -137.3838,B 24.8447,C -2.8748,E1 24.896,E2 -859.7131} C_DIS
LIN {X -19.717,Y -20.2416,Z 58,A -142.0449,B 24.8436,C -2.8852,E1 24.8865,E2 -855.0578} C_DIS
LIN {X -21.0808,Y -18.817,Z 58,A -145.775,B 24.8425,C -2.8956,E1 24.8794,E2 -851.3363} C_DIS
LIN {X -22.3449,Y -17.2971,Z 58,A -150.6193,B 24.8421,C -2.899,E1 24.871,E2 -846.4776} C_DIS
LIN {X -23.3762,Y -15.8755,Z 58,A -154.3128,B 24.8412,C -2.9069,E1 24.8651,E2 -842.7845} C_DIS
LIN {X -25.0471,Y -13.0816,Z 58,A -160.1432,B 24.8388,C -2.9291,E1 24.8571,E2 -836.9769} C_DIS
LIN {X -25.8541,Y -11.4042,Z 58,A -165.1433,B 24.8385,C -2.9317,E1 24.8513,E2 -831.9556} C_DIS
LIN {X -27.0488,Y -8.176,Z 58,A -171.5037,B 24.8358,C -2.9557,E1 24.8456,E2 -825.6163} C_DIS
LIN {X -27.5342,Y -6.3517,Z 58,A -174.6384,B 24.8341,C -2.9713,E1 24.8435,E2 -822.5008} C_DIS
LIN {X -27.8946,Y -4.5145,Z 58,A -179.1103,B 24.8332,C -2.9787,E1 24.8413,E2 -818.02} C_DIS
LIN {X -28.1495,Y -2.4658,Z 58,A 176.6585,B 24.8318,C -2.9913,E1 24.8401,E2 -813.7937} C_DIS
LIN {X -28.2578,Y -0.0449,Z 58,A 171.9966,B 24.8299,C -3.0081,E1 24.8398,E2 -809.1439} C_DIS
LIN {X -28.2102,Y 1.6332,Z 58,A 168.4841,B 24.8288,C -3.0181,E1 24.8402,E2 -805.6341} C_DIS
LIN {X -28.0223,Y 3.6349,Z 58,A 164.8467,B 24.827,C -3.0334,E1 24.8413,E2 -802.0117} C_DIS
LIN {X -27.834,Y 4.8749,Z 58,A 161.797,B 24.8265,C -3.0383,E1 24.8427,E2 -798.9555} C_DIS
LIN {X -27.323,Y 7.2061,Z 58,A 156.2811,B 24.8252,C -3.0491,E1 24.8464,E2 -793.4332} C_DIS
LIN {X -26.5027,Y 9.803,Z 58,A 151.5074,B 24.8228,C -3.0703,E1 24.8507,E2 -788.6831} C_DIS
LIN {X -25.6846,Y 11.7802,Z 58,A 147.1677,B 24.8213,C -3.083,E1 24.8555,E2 -784.35} C_DIS
LIN {X -24.8725,Y 13.4105,Z 58,A 143.3094,B 24.8202,C -3.0925,E1 24.8604,E2 -780.4938} C_DIS
LIN {X -24.0413,Y 14.8495,Z 58,A 140.192,B 24.8189,C -3.1035,E1 24.8649,E2 -777.3866} C_DIS
LIN {X -23.0764,Y 16.3086,Z 58,A 135.7743,B 24.8185,C -3.1074,E1 24.8719,E2 -772.9565} C_DIS
LIN {X -21.0841,Y 18.8133,Z 58,A 130.4937,B 24.8156,C -3.1318,E1 24.8812,E2 -767.7097} C_DIS
LIN {X -20.129,Y 19.8316,Z 58,A 127.0692,B 24.8153,C -3.1345,E1 24.8878,E2 -764.277} C_DIS
LIN {X -18.8518,Y 21.0496,Z 58,A 123.6021,B 24.8142,C -3.1433,E1 24.8949,E2 -760.8169} C_DIS
LIN {X -17.5836,Y 22.1199,Z 58,A 120.1981,B 24.8134,C -3.1502,E1 24.9023,E2 -757.4165} C_DIS
LIN {X -16.1415,Y 23.1932,Z 58,A 116.0429,B 24.813,C -3.1538,E1 24.9117,E2 -753.2553} C_DIS
LIN {X -13.9581,Y 24.5697,Z 58,A 111.4519,B 24.8113,C -3.1678,E1 24.9226,E2 -748.6838} C_DIS
LIN {X -12.9097,Y 25.1359,Z 58,A 108.2875,B 24.8115,C -3.1661,E1 24.9305,E2 -745.5065} C_DIS
LIN {X -10.1229,Y 26.3822,Z 58,A 102.4785,B 24.8101,C -3.1776,E1 24.9454,E2 -739.7117} C_DIS
LIN {X -8.3413,Y 26.9981,Z 58,A 99.088,B 24.8092,C -3.1855,E1 24.9543,E2 -736.3339} C_DIS
LIN {X -6.7028,Y 27.4509,Z 58,A 95.0564,B 24.8093,C -3.1841,E1 24.9653,E2 -732.2929} C_DIS
LIN {X -4.5213,Y 27.8933,Z 58,A 90.3362,B 24.8091,C -3.1857,E1 24.9782,E2 -727.5717} C_DIS
LIN {X -2.4291,Y 28.1532,Z 58,A 86.2937,B 24.8086,C -3.1899,E1 24.9894,E2 -723.5368} C_DIS
LIN {X 0.16,Y 28.2569,Z 58,A 80.4321,B 24.8091,C -3.1859,E1 25.0058,E2 -717.6652} C_DIS
LIN {X 2.0873,Y 28.1806,Z 58,A 76.1391,B 24.8096,C -3.1823,E1 25.0178,E2 -713.3657} C_DIS
LIN {X 6.15,Y 27.5803,Z 58,A 69.2716,B 24.8082,C -3.1933,E1 25.0366,E2 -706.5316} C_DIS
LIN {X 7.8998,Y 27.1309,Z 58,A 65.0186,B 24.8092,C -3.1852,E1 25.0481,E2 -702.2661} C_DIS
LIN {X 9.9514,Y 26.4471,Z 58,A 60.8783,B 24.8094,C -3.1839,E1 25.059,E2 -698.1311} C_DIS
LIN {X 11.6499,Y 25.7441,Z 58,A 57.2844,B 24.8097,C -3.1813,E1 25.0682,E2 -694.5398} C_DIS
LIN {X 13.3426,Y 24.9093,Z 58,A 53.2142,B 24.8106,C -3.174,E1 25.0783,E2 -690.4634} C_DIS
LIN {X 15.0215,Y 23.934,Z 58,A 49.202,B 24.8113,C -3.1675,E1 25.0879,E2 -686.4483} C_DIS
LIN {X 16.5083,Y 22.9339,Z 58,A 45.7301,B 24.8118,C -3.1633,E1 25.0958,E2 -682.9785} C_DIS
LIN {X 18.1601,Y 21.6485,Z 58,A 41.7029,B 24.8125,C -3.1581,E1 25.1046,E2 -678.954} C_DIS
LIN {X 19.2752,Y 20.663,Z 58,A 38.5758,B 24.8133,C -3.151,E1 25.111,E2 -675.8226} C_DIS
LIN {X 20.7481,Y 19.1835,Z 58,A 34.1402,B 24.8146,C -3.1397,E1 25.1196,E2 -671.3795} C_DIS
LIN {X 21.9139,Y 17.8399,Z 58,A 31.0231,B 24.8149,C -3.1372,E1 25.1252,E2 -668.2707} C_DIS
LIN {X 22.9157,Y 16.5328,Z 58,A 26.9772,B 24.8169,C -3.1211,E1 25.1319,E2 -664.2059} C_DIS
LIN {X 24.2581,Y 14.4927,Z 58,A 22.4231,B 24.8178,C -3.1132,E1 25.1387,E2 -659.6561} C_DIS
LIN {X 25.1042,Y 12.9719,Z 58,A 19.2786,B 24.8183,C -3.1084,E1 25.1428,E2 -656.5168} C_DIS
LIN {X 25.7117,Y 11.7218,Z 58,A 16.3799,B 24.8194,C -3.0997,E1 25.1463,E2 -653.6131} C_DIS
LIN {X 26.2266,Y 10.5198,Z 58,A 13.8925,B 24.82,C -3.0942,E1 25.149,E2 -651.1266} C_DIS
LIN {X 26.8146,Y 8.9147,Z 58,A 10.389,B 24.8212,C -3.0838,E1 25.1522,E2 -647.6181} C_DIS
LIN {X 27.2998,Y 7.2942,Z 58,A 6.289,B 24.8233,C -3.0656,E1 25.1553,E2 -643.4983} C_DIS
LIN {X 27.8041,Y 5.0409,Z 58,A 2.3999,B 24.8238,C -3.0612,E1 25.1575,E2 -639.6215} C_DIS
LIN {X 27.996,Y 3.8369,Z 58,A -0.9803,B 24.826,C -3.0424,E1 25.1588,E2 -636.2168} C_DIS
LIN {X 28.2513,Y 0.5902,Z 58,A -6.3099,B 24.8265,C -3.0377,E1 25.1598,E2 -630.9078} C_DIS
LIN {X 28.2457,Y -0.8144,Z 58,A -9.8086,B 24.8285,C -3.0207,E1 25.1596,E2 -627.3896} C_DIS
LIN {X 28.0985,Y -2.9921,Z 58,A -14.1894,B 24.83,C -3.0075,E1 25.1586,E2 -623.0033} C_DIS
LIN {X 27.8608,Y -4.718,Z 58,A -18.0801,B 24.8317,C -2.992,E1 25.1569,E2 -619.099} C_DIS
LIN {X 27.3081,Y -7.2633,Z 58,A -22.324,B 24.8321,C -2.9886,E1 25.1542,E2 -614.8714} C_DIS
LIN {X 26.9748,Y -8.4166,Z 58,A -26.1377,B 24.8349,C -2.9642,E1 25.151,E2 -611.0216} C_DIS
LIN {X 25.7112,Y -11.722,Z 58,A -31.8987,B 24.8353,C -2.9602,E1 25.145,E2 -605.283} C_DIS
LIN {X 25.11,Y -12.9606,Z 58,A -35.5311,B 24.8374,C -2.9418,E1 25.1404,E2 -601.6265} C_DIS
LIN {X 23.8396,Y -15.1712,Z 58,A -40.1303,B 24.8382,C -2.9343,E1 25.1339,E2 -597.0331} C_DIS
LIN {X 22.871,Y -16.5955,Z 58,A -43.8278,B 24.8395,C -2.9225,E1 25.1279,E2 -593.3256} C_DIS
LIN {X 21.2866,Y -18.5839,Z 58,A -49.4206,B 24.8415,C -2.9042,E1 25.1179,E2 -587.7152} C_DIS
LIN {X 19.6045,Y -20.3504,Z 58,A -54.0288,B 24.8424,C -2.8964,E1 25.1089,E2 -583.1081} C_DIS
LIN {X 17.789,Y -21.9551,Z 58,A -59.0639,B 24.8437,C -2.8842,E1 25.0981,E2 -578.0637} C_DIS
LIN {X 15.7872,Y -23.436,Z 58,A -63.5687,B 24.8441,C -2.8803,E1 25.0879,E2 -573.5653} C_DIS
LIN {X 14.3333,Y -24.3524,Z 58,A -67.3848,B 24.8452,C -2.8703,E1 25.0788,E2 -569.7374} C_DIS
LIN {X 12.4534,Y -25.3654,Z 58,A -71.8482,B 24.8461,C -2.8618,E1 25.0677,E2 -565.2661} C_DIS
LIN {X 9.3564,Y -26.6634,Z 58,A -79.4011,B 24.848,C -2.8448,E1 25.048,E2 -557.6895} C_DIS
LIN {X 6.8872,Y -27.4056,Z 58,A -83.5646,B 24.8474,C -2.8503,E1 25.0368,E2 -553.5458} C_DIS
LIN {X 5.1891,Y -27.7773,Z 58,A -87.0707,B 24.8477,C -2.8475,E1 25.0272,E2 -550.0373} C_DIS
LIN {X 3.4543,Y -28.0459,Z 58,A -91.1303,B 24.8484,C -2.8403,E1 25.0159,E2 -545.9639} C_DIS
LIN {X 0.7252,Y -28.2474,Z 58,A -95.8098,B 24.8478,C -2.8465,E1 25.0029,E2 -541.301} C_DIS
LIN {X 0.7252,Y -28.2474,Z 58,A -95.8098,B 24.8478,C -2.8465,E1 25.0029,E2 -541.301} C_DIS
Enddeposition()
LIN {X 0.0659,Y -27.2775,Z 58,A -94.9572,B 24.8437,C -2.884,E1 25.0056,E2 -542.2426} C_DIS
Startdeposition()
$VEL.CP = VEL_PRINT
LIN {X 3.2729,Y -27.0813,Z 58,A -89.015,B 24.8442,C -2.8794,E1 25.022,E2 -548.1706} C_DIS
LIN {X 5.2971,Y -26.7593,Z 58,A -84.4073,B 24.8435,C -2.8857,E1 25.0347,E2 -552.7884} C_DIS
LIN {X 7.2928,Y -26.2855,Z 58,A -79.5623,B 24.8424,C -2.8957,E1 25.0479,E2 -557.6495} C_DIS
LIN {X 10.5627,Y -25.1501,Z 58,A -73.4038,B 24.8427,C -2.8933,E1 25.0639,E2 -563.7893} C_DIS
LIN {X 12.0581,Y -24.4684,Z 58,A -69.6348,B 24.8417,C -2.9021,E1 25.0735,E2 -567.5693} C_DIS
LIN {X 13.6588,Y -23.612,Z 58,A -65.4523,B 24.8406,C -2.9127,E1 25.0837,E2 -571.7648} C_DIS
LIN {X 15.6726,Y -22.3267,Z 58,A -60.8795,B 24.8401,C -2.9174,E1 25.0943,E2 -576.3333} C_DIS
LIN {X 17.0779,Y -21.2711,Z 58,A -57.5238,B 24.8396,C -2.9213,E1 25.1017,E2 -579.6859} C_DIS
LIN {X 18.0522,Y -20.4503,Z 58,A -54.8966,B 24.839,C -2.9266,E1 25.1072,E2 -582.3155} C_DIS
LIN {X 18.9154,Y -19.6547,Z 58,A -52.4213,B 24.8384,C -2.9324,E1 25.1123,E2 -584.7944} C_DIS
LIN {X 19.7706,Y -18.7947,Z 58,A -49.8666,B 24.8377,C -2.9386,E1 25.1172,E2 -587.3527} C_DIS
LIN {X 20.5989,Y -17.8827,Z 58,A -47.1727,B 24.8369,C -2.9463,E1 25.1222,E2 -590.0528} C_DIS
LIN {X 21.5915,Y -16.6706,Z 58,A -43.7275,B 24.8357,C -2.9566,E1 25.1282,E2 -593.5063} C_DIS
LIN {X 22.4775,Y -15.4557,Z 58,A -40.4974,B 24.8347,C -2.9659,E1 25.1334,E2 -596.7428} C_DIS
LIN {X 23.423,Y -13.9793,Z 58,A -36.83,B 24.8335,C -2.976,E1 25.1388,E2 -600.4154} C_DIS
LIN {X 24.483,Y -12.0287,Z 58,A -32.7356,B 24.8328,C -2.9825,E1 25.1441,E2 -604.5035} C_DIS
LIN {X 25.4136,Y -9.9122,Z 58,A -26.596,B 24.8294,C -3.0126,E1 25.1507,E2 -610.6806} C_DIS
LIN {X 26.2276,Y -7.4976,Z 58,A -21.9586,B 24.8286,C -3.02,E1 25.1545,E2 -615.3092} C_DIS
LIN {X 26.6244,Y -5.9377,Z 58,A -18.7392,B 24.8276,C -3.0285,E1 25.1566,E2 -618.5299} C_DIS
LIN {X 26.938,Y -4.2965,Z 58,A -14.3993,B 24.8252,C -3.0497,E1 25.1585,E2 -622.8947} C_DIS
LIN {X 27.2774,Y -0.2942,Z 58,A -7.1223,B 24.8238,C -3.0616,E1 25.1598,E2 -630.1566} C_DIS
LIN {X 27.2669,Y 0.7639,Z 58,A -4.0786,B 24.8218,C -3.0787,E1 25.1595,E2 -633.2228} C_DIS
LIN {X 26.9733,Y 4.068,Z 58,A 2.9863,B 24.8192,C -3.1013,E1 25.1572,E2 -640.2994} C_DIS
LIN {X 26.3418,Y 7.0846,Z 58,A 8.1041,B 24.8188,C -3.1041,E1 25.154,E2 -645.3941} C_DIS
LIN {X 25.9275,Y 8.4776,Z 58,A 12.0929,B 24.8165,C -3.1243,E1 25.1506,E2 -649.4081} C_DIS
LIN {X 25.028,Y 10.8491,Z 58,A 16.9255,B 24.8154,C -3.1333,E1 25.1456,E2 -654.2355} C_DIS
LIN {X 24.2331,Y 12.5249,Z 58,A 20.9294,B 24.814,C -3.1451,E1 25.1406,E2 -658.2459} C_DIS
LIN {X 23.2124,Y 14.3284,Z 58,A 24.8475,B 24.8133,C -3.1513,E1 25.1351,E2 -662.1584} C_DIS
LIN {X 22.0372,Y 16.0768,Z 58,A 30.1184,B 24.8108,C -3.1719,E1 25.1266,E2 -667.4525} C_DIS
LIN {X 20.8121,Y 17.6341,Z 58,A 33.8032,B 24.8103,C -3.1759,E1 25.1201,E2 -671.1298} C_DIS
LIN {X 19.4985,Y 19.0768,Z 58,A 38.1344,B 24.809,C -3.1872,E1 25.1117,E2 -675.4691} C_DIS
LIN {X 18.0519,Y 20.4509,Z 58,A 41.4466,B 24.8091,C -3.1857,E1 25.105,E2 -678.7642} C_DIS
LIN {X 17.016,Y 21.3207,Z 58,A 44.8529,B 24.8078,C -3.197,E1 25.0976,E2 -682.1845} C_DIS
LIN {X 15.7109,Y 22.3001,Z 58,A 47.8854,B 24.8076,C -3.1985,E1 25.0907,E2 -685.2098} C_DIS
LIN {X 13.8006,Y 23.5298,Z 58,A 53.054,B 24.8062,C -3.2098,E1 25.0785,E2 -690.3887} C_DIS
LIN {X 12.5592,Y 24.2155,Z 58,A 55.7299,B 24.8062,C -3.2104,E1 25.0719,E2 -693.0586} C_DIS
LIN {X 11.4597,Y 24.7543,Z 58,A 58.76,B 24.8052,C -3.2181,E1 25.0642,E2 -696.0992} C_DIS
LIN {X 9.0065,Y 25.7485,Z 58,A 63.8405,B 24.8052,C -3.2185,E1 25.051,E2 -701.1695} C_DIS
LIN {X 7.9102,Y 26.1057,Z 58,A 66.4314,B 24.8048,C -3.2219,E1 25.0441,E2 -703.764} C_DIS
LIN {X 6.1272,Y 26.5811,Z 58,A 70.2221,B 24.8046,C -3.2233,E1 25.0338,E2 -707.5523} C_DIS
LIN {X 3.7642,Y 27.0173,Z 58,A 75.9747,B 24.8036,C -3.2315,E1 25.0179,E2 -713.3187} C_DIS
LIN {X 1.6132,Y 27.2304,Z 58,A 79.7308,B 24.8044,C -3.2245,E1 25.0075,E2 -717.0563} C_DIS
LIN {X 0.239,Y 27.2772,Z 58,A 82.5474,B 24.8046,C -3.2235,E1 24.9997,E2 -719.8701} C_DIS
LIN {X -1.1414,Y 27.2543,Z 58,A 85.9255,B 24.8042,C -3.2269,E1 24.9902,E2 -723.2567} C_DIS
LIN {X -2.5975,Y 27.1543,Z 58,A 88.8204,B 24.8045,C -3.224,E1 24.9822,E2 -726.146} C_DIS
LIN {X -4.422,Y 26.9174,Z 58,A 92.3889,B 24.8051,C -3.219,E1 24.9723,E2 -729.7056} C_DIS
LIN {X -5.7098,Y 26.6741,Z 58,A 95.8533,B 24.8047,C -3.2226,E1 24.9628,E2 -733.1828} C_DIS
LIN {X -8.4313,Y 25.9422,Z 58,A 101.4053,B 24.8058,C -3.2134,E1 24.948,E2 -738.7219} C_DIS
LIN {X -10.0279,Y 25.3682,Z 58,A 105.262,B 24.8061,C -3.2111,E1 24.9379,E2 -742.5811} C_DIS
LIN {X -12.0986,Y 24.4484,Z 58,A 109.6712,B 24.8073,C -3.2013,E1 24.9268,E2 -746.978} C_DIS
LIN {X -13.74,Y 23.5656,Z 58,A 113.3119,B 24.8083,C -3.1927,E1 24.918,E2 -750.6087} C_DIS
LIN {X -14.7225,Y 22.9637,Z 58,A 116.055,B 24.8086,C -3.1906,E1 24.9115,E2 -753.3555} C_DIS
LIN {X -16.2335,Y 21.9225,Z 58,A 119.7285,B 24.8096,C -3.1817,E1 24.9031,E2 -757.0206} C_DIS
LIN {X -17.3885,Y 21.0176,Z 58,A 123.1193,B 24.8101,C -3.1774,E1 24.8958,E2 -760.4137} C_DIS
LIN {X -18.5601,Y 19.9911,Z 58,A 125.9596,B 24.8114,C -3.1671,E1 24.8899,E2 -763.2409} C_DIS
LIN {X -19.4379,Y 19.1382,Z 58,A 128.6498,B 24.812,C -3.162,E1 24.8846,E2 -765.93} C_DIS
LIN {X -20.4002,Y 18.1092,Z 58,A 131.6593,B 24.8128,C -3.1551,E1 24.8789,E2 -768.9364} C_DIS
LIN {X -21.4498,Y 16.8526,Z 58,A 135.346,B 24.8137,C -3.148,E1 24.8725,E2 -772.6232} C_DIS
LIN {X -22.4897,Y 15.4379,Z 58,A 138.9704,B 24.8149,C -3.1378,E1 24.8666,E2 -776.2409} C_DIS
LIN {X -23.5149,Y 13.8258,Z 58,A 143.6089,B 24.8157,C -3.1306,E1 24.8599,E2 -780.8862} C_DIS
LIN {X -24.8368,Y 11.28,Z 58,A 149.7113,B 24.8177,C -3.1137,E1 24.8524,E2 -786.9811} C_DIS
LIN {X -25.7249,Y 9.0737,Z 58,A 153.7517,B 24.8201,C -3.093,E1 24.8484,E2 -790.9945} C_DIS
LIN {X -26.4319,Y 6.742,Z 58,A 160.548,B 24.8208,C -3.0876,E1 24.8434,E2 -797.8172} C_DIS
LIN {X -27.0913,Y 3.1873,Z 58,A 167.4999,B 24.824,C -3.06,E1 24.8404,E2 -804.7445} C_DIS
LIN {X -27.2492,Y 1.2606,Z 58,A 170.71,B 24.826,C -3.0422,E1 24.8399,E2 -807.9314} C_DIS
LIN {X -27.2792,Y -0.2018,Z 58,A 174.29,B 24.8268,C -3.0357,E1 24.8399,E2 -811.5173} C_DIS
LIN {X -27.1971,Y -2.1014,Z 58,A 178.0054,B 24.8284,C -3.0217,E1 24.8404,E2 -815.2214} C_DIS
LIN {X -27.0533,Y -3.4953,Z 58,A -179.0034,B 24.8294,C -3.0129,E1 24.8414,E2 -818.2096} C_DIS
LIN {X -26.8249,Y -4.9505,Z 58,A -175.7089,B 24.8303,C -3.0048,E1 24.843,E2 -821.5041} C_DIS
LIN {X -26.4342,Y -6.7331,Z 58,A -171.7241,B 24.8315,C -2.9943,E1 24.8456,E2 -825.487} C_DIS
LIN {X -25.8092,Y -8.8318,Z 58,A -167.5258,B 24.8333,C -2.9784,E1 24.8491,E2 -829.6715} C_DIS
LIN {X -25.2981,Y -10.2035,Z 58,A -164.1624,B 24.8341,C -2.9715,E1 24.8525,E2 -833.0373} C_DIS
LIN {X -24.508,Y -11.9783,Z 58,A -160.5481,B 24.8356,C -2.9573,E1 24.8567,E2 -836.6374} C_DIS
LIN {X -23.9816,Y -12.9989,Z 58,A -157.9445,B 24.8362,C -2.9522,E1 24.8601,E2 -839.2425} C_DIS
LIN {X -23.1777,Y -14.3839,Z 58,A -153.9326,B 24.8367,C -2.9478,E1 24.8658,E2 -843.2648} C_DIS
LIN {X -22.2528,Y -15.7771,Z 58,A -150.5053,B 24.8377,C -2.9387,E1 24.8713,E2 -846.6871} C_DIS
LIN {X -20.9899,Y -17.4219,Z 58,A -146.2787,B 24.8389,C -2.9278,E1 24.8786,E2 -850.9074} C_DIS
LIN {X -19.8803,Y -18.6781,Z 58,A -142.9393,B 24.8399,C -2.919,E1 24.8849,E2 -854.2405} C_DIS
LIN {X -18.9972,Y -19.5759,Z 58,A -139.9888,B 24.8402,C -2.9158,E1 24.8908,E2 -857.1957} C_DIS
LIN {X -17.9115,Y -20.5738,Z 58,A -136.8799,B 24.8409,C -2.91,E1 24.8973,E2 -860.3031} C_DIS
LIN {X -16.3055,Y -21.8687,Z 58,A -132.5199,B 24.8417,C -2.9027,E1 24.9069,E2 -864.6615} C_DIS
LIN {X -14.5963,Y -23.045,Z 58,A -128.852,B 24.843,C -2.8906,E1 24.9154,E2 -868.3129} C_DIS
LIN {X -13.1895,Y -23.8778,Z 58,A -124.2516,B 24.8425,C -2.8952,E1 24.9266,E2 -872.9376} C_DIS
LIN {X -11.0693,Y -24.9311,Z 58,A -119.7332,B 24.8435,C -2.8859,E1 24.938,E2 -877.4453} C_DIS
LIN {X -9.1504,Y -25.698,Z 58,A -115.66,B 24.8442,C -2.8798,E1 24.9486,E2 -881.5124} C_DIS
LIN {X -6.8392,Y -26.4069,Z 58,A -109.5528,B 24.8436,C -2.8855,E1 24.9651,E2 -887.643} C_DIS
LIN {X -4.5244,Y -26.9004,Z 58,A -104.8266,B 24.844,C -2.8816,E1 24.978,E2 -892.3648} C_DIS
LIN {X -1.5752,Y -27.2324,Z 58,A -99.1175,B 24.8445,C -2.8764,E1 24.9939,E2 -898.0643} C_DIS
LIN {X 0.0659,Y -27.2775,Z 58,A -94.9571,B 24.8437,C -2.8839,E1 25.0056,E2 -902.2426} C_DIS
Enddeposition()
LIN {X 0.0659,Y -27.2775,Z 58,A -94.9571,B 24.8437,C -2.8839,E1 25.0056,E2 -902.2426} C_DIS
Startdeposition()
$VEL.CP = VEL_PRINT
LIN {X -0.4263,Y -26.2956,Z 58,A -98.4219,B 24.8443,C -2.8783,E1 24.9959,E2 -898.7646} C_DIS
LIN {X -1.9073,Y -26.2301,Z 58,A -101.9097,B 24.8446,C -2.8759,E1 24.9861,E2 -895.2701} C_DIS
LIN {X -3.656,Y -26.0437,Z 58,A -105.7946,B 24.8446,C -2.8761,E1 24.9753,E2 -891.3828} C_DIS
LIN {X -5.3554,Y -25.748,Z 58,A -109.8647,B 24.8447,C -2.8749,E1 24.9642,E2 -887.3055} C_DIS
LIN {X -7.6976,Y -25.1474,Z 58,A -114.5796,B 24.8439,C -2.8825,E1 24.9515,E2 -882.6014} C_DIS
LIN {X -8.957,Y -24.7268,Z 58,A -118.0276,B 24.8441,C -2.8806,E1 24.9424,E2 -879.1421} C_DIS
LIN {X -11.419,Y -23.6906,Z 58,A -123.6574,B 24.8433,C -2.8882,E1 24.928,E2 -873.5169} C_DIS
LIN {X -12.9085,Y -22.913,Z 58,A -126.9533,B 24.8425,C -2.8956,E1 24.92,E2 -870.2292} C_DIS
LIN {X -14.2928,Y -22.0763,Z 58,A -130.901,B 24.8422,C -2.8977,E1 24.9106,E2 -866.2742} C_DIS
LIN {X -16.2667,Y -20.6648,Z 58,A -136.4228,B 24.8414,C -2.905,E1 24.8983,E2 -860.7502} C_DIS
LIN {X -17.7305,Y -19.423,Z 58,A -140.3837,B 24.8404,C -2.9145,E1 24.89,E2 -856.796} C_DIS
LIN {X -19.1752,Y -17.9987,Z 58,A -144.55,B 24.8392,C -2.9252,E1 24.8819,E2 -852.6378} C_DIS
LIN {X -20.0772,Y -16.9868,Z 58,A -147.3967,B 24.8384,C -2.9324,E1 24.8766,E2 -849.7953} C_DIS
LIN {X -20.8808,Y -15.9886,Z 58,A -150.2597,B 24.8377,C -2.9385,E1 24.8717,E2 -846.9332} C_DIS
LIN {X -21.8273,Y -14.6702,Z 58,A -154.7228,B 24.8374,C -2.9415,E1 24.8646,E2 -842.4553} C_DIS
LIN {X -23.4064,Y -11.9905,Z 58,A -160.9482,B 24.8351,C -2.9625,E1 24.8562,E2 -836.2475} C_DIS
LIN {X -24.2732,Y -10.122,Z 58,A -165.4822,B 24.8337,C -2.9746,E1 24.8511,E2 -831.7175} C_DIS
LIN {X -24.8373,Y -8.6458,Z 58,A -168.5716,B 24.8324,C -2.9864,E1 24.8481,E2 -828.639} C_DIS
LIN {X -25.2734,Y -7.2736,Z 58,A -171.8829,B 24.8315,C -2.9946,E1 24.8454,E2 -825.3281} C_DIS
LIN {X -25.7373,Y -5.4058,Z 58,A -176.6822,B 24.8304,C -3.0038,E1 24.8425,E2 -820.5227} C_DIS
LIN {X -26.0974,Y -3.2527,Z 58,A 178.608,B 24.8287,C -3.0186,E1 24.8406,E2 -815.8202} C_DIS
LIN {X -26.282,Y -0.9542,Z 58,A 174.1647,B 24.8266,C -3.0372,E1 24.8398,E2 -811.3949} C_DIS
LIN {X -26.2939,Y 0.5197,Z 58,A 170.8646,B 24.8255,C -3.0468,E1 24.8398,E2 -808.0977} C_DIS
LIN {X -26.2263,Y 1.9586,Z 58,A 167.4954,B 24.8245,C -3.0553,E1 24.8404,E2 -804.7287} C_DIS
LIN {X -26.0185,Y 3.8302,Z 58,A 163.5683,B 24.8229,C -3.069,E1 24.8418,E2 -800.811} C_DIS
LIN {X -25.7499,Y 5.3457,Z 58,A 160.1787,B 24.8218,C -3.0792,E1 24.8436,E2 -797.4258} C_DIS
LIN {X -25.3165,Y 7.1201,Z 58,A 155.4877,B 24.8208,C -3.0876,E1 24.8469,E2 -792.7275} C_DIS
LIN {X -24.6514,Y 9.1635,Z 58,A 150.9341,B 24.8191,C -3.1023,E1 24.8512,E2 -788.1833} C_DIS
LIN {X -23.8582,Y 11.0636,Z 58,A 147.3537,B 24.8169,C -3.1205,E1 24.8551,E2 -784.6268} C_DIS
LIN {X -23.3752,Y 12.0519,Z 58,A 143.9203,B 24.8168,C -3.1216,E1 24.8595,E2 -781.1775} C_DIS
LIN {X -22.2319,Y 14.05,Z 58,A 139.9114,B 24.8145,C -3.1412,E1 24.8652,E2 -777.1949} C_DIS
LIN {X -21.425,Y 15.2516,Z 58,A 136.1841,B 24.8139,C -3.1463,E1 24.8711,E2 -773.4614} C_DIS
LIN {X -20.6391,Y 16.2992,Z 58,A 132.9288,B 24.8133,C -3.1513,E1 24.8766,E2 -770.2027} C_DIS
LIN {X -19.2052,Y 17.9667,Z 58,A 128.3527,B 24.8117,C -3.1643,E1 24.8852,E2 -765.6374} C_DIS
LIN {X -17.7351,Y 19.4193,Z 58,A 124.1037,B 24.8103,C -3.1762,E1 24.8937,E2 -761.3993} C_DIS
LIN {X -16.3146,Y 20.6269,Z 58,A 119.707,B 24.8095,C -3.1828,E1 24.9032,E2 -757.0014} C_DIS
LIN {X -14.9304,Y 21.6502,Z 58,A 116.127,B 24.8085,C -3.1912,E1 24.9113,E2 -753.4293} C_DIS
LIN {X -13.4101,Y 22.6232,Z 58,A 111.568,B 24.8081,C -3.1941,E1 24.9222,E2 -748.8631} C_DIS
LIN {X -11.282,Y 23.7562,Z 58,A 107.0137,B 24.8065,C -3.2072,E1 24.9335,E2 -744.3278} C_DIS
LIN {X -9.8173,Y 24.3982,Z 58,A 103.7293,B 24.8058,C -3.2135,E1 24.9419,E2 -741.0508} C_DIS
LIN {X -8.2997,Y 24.9553,Z 58,A 99.5437,B 24.8058,C -3.2129,E1 24.9529,E2 -736.8557} C_DIS
LIN {X -6.0453,Y 25.5951,Z 58,A 95.3586,B 24.8044,C -3.2249,E1 24.9642,E2 -732.6928} C_DIS
LIN {X -4.1381,Y 25.9713,Z 58,A 89.9145,B 24.8051,C -3.2187,E1 24.9792,E2 -727.2284} C_DIS
LIN {X -2.2748,Y 26.2008,Z 58,A 86.7002,B 24.804,C -3.2278,E1 24.988,E2 -724.0338} C_DIS
LIN {X -0.8114,Y 26.2865,Z 58,A 82.7698,B 24.8047,C -3.2228,E1 24.999,E2 -720.0907} C_DIS
LIN {X 1.6409,Y 26.2477,Z 58,A 77.8798,B 24.8041,C -3.2271,E1 25.0127,E2 -715.212} C_DIS
LIN {X 3.4525,Y 26.0715,Z 58,A 73.6738,B 24.8045,C -3.2243,E1 25.0243,E2 -711.0026} C_DIS
LIN {X 5.2134,Y 25.7772,Z 58,A 70.1012,B 24.8043,C -3.2257,E1 25.0341,E2 -707.4373} C_DIS
LIN {X 7.0893,Y 25.3253,Z 58,A 65.2403,B 24.8053,C -3.2172,E1 25.0473,E2 -702.5637} C_DIS
LIN {X 9.2734,Y 24.6098,Z 58,A 60.5489,B 24.8055,C -3.2159,E1 25.0596,E2 -697.8786} C_DIS
LIN {X 11.2692,Y 23.7626,Z 58,A 56.6477,B 24.8052,C -3.2187,E1 25.0695,E2 -693.9936} C_DIS
LIN {X 12.3833,Y 23.2016,Z 58,A 53.0246,B 24.8066,C -3.2064,E1 25.0786,E2 -690.3513} C_DIS
LIN {X 14.0533,Y 22.2296,Z 58,A 49.5065,B 24.8066,C -3.2072,E1 25.0869,E2 -686.8461} C_DIS
LIN {X 15.2612,Y 21.4181,Z 58,A 45.755,B 24.8079,C -3.1962,E1 25.0956,E2 -683.0813} C_DIS
LIN {X 16.6913,Y 20.3233,Z 58,A 42.35,B 24.8081,C -3.1946,E1 25.103,E2 -679.6852} C_DIS
LIN {X 17.7053,Y 19.4466,Z 58,A 39.2635,B 24.809,C -3.1872,E1 25.1095,E2 -676.5935} C_DIS
LIN {X 19.1192,Y 18.0581,Z 58,A 34.3619,B 24.8108,C -3.172,E1 25.1191,E2 -671.6768} C_DIS
LIN {X 20.4203,Y 16.5721,Z 58,A 30.0036,B 24.812,C -3.1617,E1 25.1269,E2 -667.314} C_DIS
LIN {X 22.1945,Y 14.1087,Z 58,A 23.8363,B 24.8134,C -3.1503,E1 25.1366,E2 -661.1501} C_DIS
LIN {X 23.3537,Y 12.0939,Z 58,A 18.3642,B 24.8155,C -3.1324,E1 25.1439,E2 -655.6643} C_DIS
LIN {X 24.3869,Y 9.8441,Z 58,A 13.5553,B 24.8165,C -3.124,E1 25.1492,E2 -650.8619} C_DIS
LIN {X 25.0386,Y 8.0441,Z 58,A 9.6223,B 24.8176,C -3.1148,E1 25.1528,E2 -646.929} C_DIS
LIN {X 25.6636,Y 5.7482,Z 58,A 3.5194,B 24.8206,C -3.0888,E1 25.1569,E2 -640.7997} C_DIS
LIN {X 26.0909,Y 3.3027,Z 58,A -1.402,B 24.8219,C -3.0779,E1 25.1589,E2 -635.8815} C_DIS
LIN {X 26.283,Y 0.9176,Z 58,A -5.7809,B 24.8226,C -3.0715,E1 25.1597,E2 -631.5135} C_DIS
LIN {X 26.2951,Y -0.4553,Z 58,A -9.2953,B 24.8244,C -3.056,E1 25.1597,E2 -627.9834} C_DIS
LIN {X 26.1491,Y -2.8047,Z 58,A -14.7622,B 24.8267,C -3.036,E1 25.1584,E2 -622.5016} C_DIS
LIN {X 25.8594,Y -4.788,Z 58,A -18.566,B 24.8275,C -3.029,E1 25.1567,E2 -618.7035} C_DIS
LIN {X 25.581,Y -6.1048,Z 58,A -21.6613,B 24.8288,C -3.0181,E1 25.1547,E2 -615.6002} C_DIS
LIN {X 25.1793,Y -7.5921,Z 58,A -24.463,B 24.8292,C -3.0143,E1 25.1526,E2 -612.8055} C_DIS
LIN {X 24.5345,Y -9.472,Z 58,A -29.8464,B 24.8321,C -2.989,E1 25.1474,E2 -607.3924} C_DIS
LIN {X 23.7221,Y -11.3535,Z 58,A -33.2307,B 24.8321,C -2.9884,E1 25.1435,E2 -604.0251} C_DIS
LIN {X 22.6551,Y -13.3561,Z 58,A -39.545,B 24.8355,C -2.9588,E1 25.1348,E2 -597.6735} C_DIS
LIN {X 21.2394,Y -15.509,Z 58,A -44.4335,B 24.8362,C -2.9519,E1 25.127,E2 -592.7924} C_DIS
LIN {X 19.9066,Y -17.1868,Z 58,A -48.982,B 24.8374,C -2.9413,E1 25.1189,E2 -588.2399} C_DIS
LIN {X 18.278,Y -18.9091,Z 58,A -54.5003,B 24.8392,C -2.9252,E1 25.108,E2 -582.7069} C_DIS
LIN {X 16.3826,Y -20.5733,Z 58,A -59.4521,B 24.8399,C -2.9191,E1 25.0975,E2 -577.7596} C_DIS
LIN {X 14.7047,Y -21.804,Z 58,A -63.9507,B 24.8408,C -2.9105,E1 25.0872,E2 -573.2562} C_DIS
LIN {X 13.0068,Y -22.8574,Z 58,A -68.2673,B 24.8416,C -2.9031,E1 25.0768,E2 -568.9353} C_DIS
LIN {X 11.5912,Y -23.607,Z 58,A -71.4702,B 24.8419,C -2.9004,E1 25.0689,E2 -565.7347} C_DIS
LIN {X 10.3555,Y -24.1746,Z 58,A -74.3629,B 24.8423,C -2.8967,E1 25.0615,E2 -562.8405} C_DIS
LIN {X 8.4678,Y -24.8986,Z 58,A -79.6002,B 24.8438,C -2.8829,E1 25.0477,E2 -557.5811} C_DIS
LIN {X 6.5846,Y -25.4613,Z 58,A -83.024,B 24.8434,C -2.8866,E1 25.0385,E2 -554.1719} C_DIS
LIN {X 5.5521,Y -25.7063,Z 58,A -85.6035,B 24.8439,C -2.882,E1 25.0314,E2 -551.5848} C_DIS
LIN {X 3.6508,Y -26.0444,Z 58,A -89.4702,B 24.8439,C -2.8821,E1 25.0208,E2 -547.7223} C_DIS
LIN {X 2.0628,Y -26.218,Z 58,A -93.4171,B 24.8446,C -2.876,E1 25.0098,E2 -543.7633} C_DIS
LIN {X 0.3688,Y -26.2966,Z 58,A -96.892,B 24.8446,C -2.8768,E1 25.0001,E2 -540.291} C_DIS
LIN {X 0.3688,Y -26.2966,Z 58,A -96.892,B 24.8446,C -2.8768,E1 25.0001,E2 -540.291} C_DIS
Enddeposition()
LIN {X 0.0546,Y -25.3146,Z 58,A -96.1598,B 24.8413,C -2.9062,E1 25.0023,E2 -541.0931} C_DIS
Startdeposition()
$VEL.CP = VEL_PRINT
LIN {X 2.1176,Y -25.2311,Z 58,A -91.2062,B 24.8408,C -2.9105,E1 25.0162,E2 -546.0551} C_DIS
LIN {X 3.3676,Y -25.0948,Z 58,A -88.3552,B 24.8406,C -2.9123,E1 25.0241,E2 -548.9082} C_DIS
LIN {X 5.225,Y -24.7752,Z 58,A -83.767,B 24.8399,C -2.9188,E1 25.0367,E2 -553.5064} C_DIS
LIN {X 6.9295,Y -24.3532,Z 58,A -79.7965,B 24.8395,C -2.9229,E1 25.0474,E2 -557.4803} C_DIS
LIN {X 9.0075,Y -23.6631,Z 58,A -75.0977,B 24.8391,C -2.9266,E1 25.0598,E2 -562.1783} C_DIS
LIN {X 10.7817,Y -22.9098,Z 58,A -70.9372,B 24.8386,C -2.931,E1 25.0704,E2 -566.3391} C_DIS
LIN {X 11.9372,Y -22.3296,Z 58,A -68.1489,B 24.8382,C -2.9344,E1 25.0773,E2 -569.1277} C_DIS
LIN {X 13.0316,Y -21.7093,Z 58,A -65.1474,B 24.8375,C -2.941,E1 25.0845,E2 -572.1358} C_DIS
LIN {X 14.0858,Y -21.0405,Z 58,A -62.5486,B 24.8371,C -2.944,E1 25.0906,E2 -574.7332} C_DIS
LIN {X 15.1223,Y -20.3081,Z 58,A -59.5126,B 24.8363,C -2.9515,E1 25.0975,E2 -577.7763} C_DIS
LIN {X 16.3052,Y -19.3713,Z 58,A -55.9491,B 24.8353,C -2.9605,E1 25.1052,E2 -581.3475} C_DIS
LIN {X 17.5282,Y -18.2719,Z 58,A -52.3524,B 24.8345,C -2.9676,E1 25.1126,E2 -584.9465} C_DIS
LIN {X 18.6731,Y -17.1,Z 58,A -48.6421,B 24.8335,C -2.9766,E1 25.1197,E2 -588.662} C_DIS
LIN {X 19.675,Y -15.9371,Z 58,A -45.2172,B 24.8325,C -2.9849,E1 25.1258,E2 -592.0907} C_DIS
LIN {X 20.7248,Y -14.5461,Z 58,A -41.3978,B 24.8315,C -2.994,E1 25.1321,E2 -595.9132} C_DIS
LIN {X 21.4274,Y -13.4895,Z 58,A -38.1025,B 24.8301,C -3.0067,E1 25.1371,E2 -599.2221} C_DIS
LIN {X 22.4748,Y -11.6612,Z 58,A -33.5934,B 24.8289,C -3.0172,E1 25.1432,E2 -603.7326} C_DIS
LIN {X 23.2195,Y -10.0965,Z 58,A -29.3821,B 24.8272,C -3.0321,E1 25.148,E2 -607.9563} C_DIS
LIN {X 24.0615,Y -7.8835,Z 58,A -24.6335,B 24.8261,C -3.0411,E1 25.1525,E2 -612.6997} C_DIS
LIN {X 24.5306,Y -6.2727,Z 58,A -20.5043,B 24.8244,C -3.0566,E1 25.1555,E2 -616.8419} C_DIS
LIN {X 24.9458,Y -4.3385,Z 58,A -16.6395,B 24.8236,C -3.0634,E1 25.1577,E2 -620.7001} C_DIS
LIN {X 25.121,Y -3.1677,Z 58,A -13.6248,B 24.8222,C -3.0757,E1 25.1588,E2 -623.7261} C_DIS
LIN {X 25.2707,Y -1.5796,Z 58,A -9.8079,B 24.8206,C -3.0894,E1 25.1596,E2 -627.5528} C_DIS
LIN {X 25.3206,Y 0.1111,Z 58,A -6.0028,B 24.8192,C -3.101,E1 25.1597,E2 -631.3628} C_DIS
LIN {X 25.2227,Y 2.2189,Z 58,A -0.9383,B 24.8171,C -3.1192,E1 25.1588,E2 -636.4403} C_DIS
LIN {X 24.9464,Y 4.3326,Z 58,A 3.6944,B 24.8156,C -3.1317,E1 25.1568,E2 -641.0753} C_DIS
LIN {X 24.4526,Y 6.5698,Z 58,A 8.3518,B 24.8145,C -3.1411,E1 25.1537,E2 -645.728} C_DIS
LIN {X 24.0702,Y 7.8564,Z 58,A 11.9274,B 24.8127,C -3.1561,E1 25.1507,E2 -649.3189} C_DIS
LIN {X 23.1161,Y 10.3317,Z 58,A 17.425,B 24.8114,C -3.1672,E1 25.1449,E2 -654.8125} C_DIS
LIN {X 22.5877,Y 11.4399,Z 58,A 20.2657,B 24.8104,C -3.1754,E1 25.1414,E2 -657.6576} C_DIS
LIN {X 21.5836,Y 13.2384,Z 58,A 25.1136,B 24.8087,C -3.1895,E1 25.1346,E2 -662.5139} C_DIS
LIN {X 20.7123,Y 14.5638,Z 58,A 28.6863,B 24.8076,C -3.1981,E1 25.1289,E2 -666.0895} C_DIS
LIN {X 19.4164,Y 16.2513,Z 58,A 33.0063,B 24.8069,C -3.2039,E1 25.1214,E2 -670.4031} C_DIS
LIN {X 18.3942,Y 17.3997,Z 58,A 36.7987,B 24.8056,C -3.2148,E1 25.1142,E2 -674.2045} C_DIS
LIN {X 17.393,Y 18.4006,Z 58,A 39.5436,B 24.8054,C -3.2165,E1 25.1088,E2 -676.9419} C_DIS
LIN {X 16.4272,Y 19.2677,Z 58,A 43.0654,B 24.804,C -3.2281,E1 25.1013,E2 -680.4774} C_DIS
LIN {X 14.8562,Y 20.5027,Z 58,A 47.19,B 24.8035,C -3.2319,E1 25.0922,E2 -684.596} C_DIS
LIN {X 12.9499,Y 21.7573,Z 58,A 53.5777,B 24.8011,C -3.2517,E1 25.077,E2 -691.0106} C_DIS
LIN {X 10.8537,Y 22.8758,Z 58,A 58.4419,B 24.8009,C -3.2531,E1 25.0648,E2 -695.8652} C_DIS
LIN {X 8.4429,Y 23.8708,Z 58,A 63.7715,B 24.8009,C -3.2533,E1 25.051,E2 -701.1835} C_DIS
LIN {X 6.6368,Y 24.4346,Z 58,A 68.1187,B 24.8005,C -3.2568,E1 25.0393,E2 -705.5317} C_DIS
LIN {X 4.7219,Y 24.8757,Z 58,A 72.8236,B 24.8,C -3.2611,E1 25.0264,E2 -710.2408} C_DIS
LIN {X 2.6487,Y 25.1809,Z 58,A 77.2518,B 24.8002,C -3.2594,E1 25.0142,E2 -714.6613} C_DIS
LIN {X 0.875,Y 25.3049,Z 58,A 81.2392,B 24.8002,C -3.2589,E1 25.0031,E2 -718.6463} C_DIS
LIN {X -0.7588,Y 25.3085,Z 58,A 84.9044,B 24.8004,C -3.2578,E1 24.9928,E2 -722.3089} C_DIS
LIN {X -2.2681,Y 25.2181,Z 58,A 88.1825,B 24.8007,C -3.2552,E1 24.9837,E2 -725.5822} C_DIS
LIN {X -3.9357,Y 25.0122,Z 58,A 92.4618,B 24.8005,C -3.2565,E1 24.9719,E2 -729.8681} C_DIS
LIN {X -5.635,Y 24.6849,Z 58,A 95.9888,B 24.8013,C -3.2503,E1 24.9623,E2 -733.3846} C_DIS
LIN {X -7.0587,Y 24.3162,Z 58,A 99.3014,B 24.8017,C -3.2468,E1 24.9534,E2 -736.694} C_DIS
LIN {X -8.4307,Y 23.8751,Z 58,A 103.0049,B 24.8017,C -3.2462,E1 24.9436,E2 -740.4029} C_DIS
LIN {X -10.4589,Y 23.0584,Z 58,A 107.4446,B 24.8031,C -3.2357,E1 24.9322,E2 -744.828} C_DIS
LIN {X -11.669,Y 22.47,Z 58,A 110.3335,B 24.8038,C -3.2299,E1 24.925,E2 -747.7106} C_DIS
LIN {X -13.0234,Y 21.7142,Z 58,A 113.7777,B 24.8046,C -3.2234,E1 24.9167,E2 -751.1495} C_DIS
LIN {X -14.1301,Y 21.0105,Z 58,A 117.204,B 24.8049,C -3.2209,E1 24.9086,E2 -754.5809} C_DIS
LIN {X -15.5964,Y 19.9458,Z 58,A 121.6936,B 24.8056,C -3.2151,E1 24.8986,E2 -759.0726} C_DIS
LIN {X -16.9911,Y 18.7724,Z 58,A 125.878,B 24.8067,C -3.2063,E1 24.8899,E2 -763.2527} C_DIS
LIN {X -18.5079,Y 17.2789,Z 58,A 130.4493,B 24.8082,C -3.1934,E1 24.881,E2 -767.8127} C_DIS
LIN {X -19.8261,Y 15.7488,Z 58,A 135.1001,B 24.8095,C -3.1824,E1 24.8727,E2 -772.4586} C_DIS
LIN {X -21.0146,Y 14.1238,Z 58,A 139.6244,B 24.811,C -3.1701,E1 24.8655,E2 -776.9757} C_DIS
LIN {X -21.8801,Y 12.7422,Z 58,A 143.1545,B 24.8123,C -3.159,E1 24.8604,E2 -780.4974} C_DIS
LIN {X -22.5162,Y 11.5809,Z 58,A 145.9267,B 24.8135,C -3.1492,E1 24.8568,E2 -783.2609} C_DIS
LIN {X -23.1683,Y 10.2144,Z 58,A 149.9399,B 24.8143,C -3.1425,E1 24.8521,E2 -787.2798} C_DIS
LIN {X -23.9251,Y 8.2883,Z 58,A 154.6032,B 24.816,C -3.1284,E1 24.8476,E2 -791.9356} C_DIS
LIN {X -24.6331,Y 5.8575,Z 58,A 160.9405,B 24.8177,C -3.1141,E1 24.8431,E2 -798.2757} C_DIS
LIN {X -25.0452,Y 3.7186,Z 58,A 165.1115,B 24.8199,C -3.0948,E1 24.8412,E2 -802.4251} C_DIS
LIN {X -25.231,Y 2.1218,Z 58,A 168.8988,B 24.8212,C -3.0842,E1 24.8401,E2 -806.2099} C_DIS
LIN {X -25.3178,Y 0.3419,Z 58,A 172.527,B 24.8229,C -3.0695,E1 24.8398,E2 -809.8247} C_DIS
LIN {X -25.3075,Y -0.7919,Z 58,A 175.8577,B 24.8233,C -3.0656,E1 24.84,E2 -813.1661} C_DIS
LIN {X -25.085,Y -3.4418,Z 58,A -178.33,B 24.8256,C -3.046,E1 24.8417,E2 -818.9662} C_DIS
LIN {X -24.7413,Y -5.3816,Z 58,A -173.7866,B 24.8271,C -3.033,E1 24.8442,E2 -823.5054} C_DIS
LIN {X -24.2472,Y -7.2909,Z 58,A -169.4514,B 24.8287,C -3.0192,E1 24.8474,E2 -827.8326} C_DIS
LIN {X -23.6016,Y -9.1688,Z 58,A -164.6911,B 24.83,C -3.0079,E1 24.852,E2 -832.5927} C_DIS
LIN {X -22.8864,Y -10.8317,Z 58,A -160.8564,B 24.8314,C -2.9951,E1 24.8564,E2 -836.4179} C_DIS
LIN {X -22.1742,Y -12.2225,Z 58,A -157.0844,B 24.8323,C -2.9871,E1 24.8614,E2 -840.1908} C_DIS
LIN {X -21.1173,Y -13.9698,Z 58,A -152.8399,B 24.8339,C -2.9732,E1 24.8676,E2 -844.4237} C_DIS
LIN {X -20.136,Y -15.351,Z 58,A -148.4577,B 24.8345,C -2.9675,E1 24.8749,E2 -848.8132} C_DIS
LIN {X -18.9869,Y -16.7514,Z 58,A -144.8437,B 24.8359,C -2.9553,E1 24.8814,E2 -852.4146} C_DIS
LIN {X -18.0705,Y -17.7356,Z 58,A -141.9839,B 24.8367,C -2.9477,E1 24.8869,E2 -855.2687} C_DIS
LIN {X -17.3299,Y -18.4599,Z 58,A -139.5127,B 24.8371,C -2.9439,E1 24.8919,E2 -857.7409} C_DIS
LIN {X -16.5132,Y -19.1943,Z 58,A -136.0721,B 24.8369,C -2.9456,E1 24.8992,E2 -861.199} C_DIS
LIN {X -14.1882,Y -20.9709,Z 58,A -130.1099,B 24.8387,C -2.9301,E1 24.9126,E2 -867.1451} C_DIS
LIN {X -12.3279,Y -22.116,Z 58,A -124.8871,B 24.8392,C -2.9252,E1 24.9252,E2 -872.372} C_DIS
LIN {X -10.5078,Y -23.0365,Z 58,A -120.3301,B 24.8398,C -2.9194,E1 24.9367,E2 -876.9271} C_DIS
LIN {X -8.7635,Y -23.7551,Z 58,A -116.0696,B 24.8403,C -2.9154,E1 24.9478,E2 -881.1871} C_DIS
LIN {X -6.9007,Y -24.3613,Z 58,A -111.948,B 24.8409,C -2.9099,E1 24.9587,E2 -885.3026} C_DIS
LIN {X -5.5509,Y -24.7039,Z 58,A -108.6819,B 24.8409,C -2.9093,E1 24.9676,E2 -888.5716} C_DIS
LIN {X -3.9693,Y -25.0068,Z 58,A -105.0118,B 24.8411,C -2.9083,E1 24.9777,E2 -892.2431} C_DIS
LIN {X -2.1961,Y -25.2248,Z 58,A -100.7558,B 24.8409,C -2.9097,E1 24.9895,E2 -896.5049} C_DIS
LIN {X -0.2617,Y -25.3187,Z 58,A -96.1738,B 24.8407,C -2.9121,E1 25.0023,E2 -901.0931} C_DIS
LIN {X -0.2617,Y -25.3187,Z 58,A -96.1738,B 24.8407,C -2.9121,E1 25.0023,E2 -901.0931} C_DIS
Enddeposition()
LIN {X 0.0345,Y -24.3378,Z 58,A -95.7619,B 24.839,C -2.9266,E1 25.0036,E2 -901.5396} C_DIS
Startdeposition()
$VEL.CP = VEL_PRINT
LIN {X -0.7385,Y -24.3295,Z 58,A -99.4411,B 24.8408,C -2.9108,E1 24.9932,E2 -897.8227} C_DIS
LIN {X -2.2428,Y -24.2371,Z 58,A -103.0723,B 24.8408,C -2.9102,E1 24.9831,E2 -894.1884} C_DIS
LIN {X -4.0989,Y -23.9932,Z 58,A -108.0444,B 24.8412,C -2.9069,E1 24.9693,E2 -889.2043} C_DIS
LIN {X -5.9419,Y -23.6046,Z 58,A -112.8222,B 24.8412,C -2.9067,E1 24.9564,E2 -884.4193} C_DIS
LIN {X -8.5697,Y -22.7822,Z 58,A -118.2729,B 24.8399,C -2.9191,E1 24.942,E2 -878.9879} C_DIS
LIN {X -9.7596,Y -22.2984,Z 58,A -121.4562,B 24.8397,C -2.921,E1 24.9338,E2 -875.802} C_DIS
LIN {X -11.1928,Y -21.6149,Z 58,A -124.7133,B 24.8388,C -2.9286,E1 24.9257,E2 -872.5546} C_DIS
LIN {X -12.4257,Y -20.9301,Z 58,A -128.3931,B 24.8386,C -2.9307,E1 24.9167,E2 -868.8689} C_DIS
LIN {X -13.7376,Y -20.0938,Z 58,A -132.3688,B 24.8382,C -2.9343,E1 24.9074,E2 -864.8887} C_DIS
LIN {X -15.1042,Y -19.0875,Z 58,A -136.4075,B 24.8375,C -2.9409,E1 24.8985,E2 -860.8511} C_DIS
LIN {X -16.2951,Y -18.0816,Z 58,A -140.0824,B 24.8367,C -2.9478,E1 24.8908,E2 -857.1783} C_DIS
LIN {X -17.5674,Y -16.8481,Z 58,A -143.8466,B 24.8355,C -2.9587,E1 24.8833,E2 -853.4242} C_DIS
LIN {X -18.2885,Y -16.0624,Z 58,A -146.6688,B 24.8351,C -2.9624,E1 24.8781,E2 -850.5982} C_DIS
LIN {X -19.3564,Y -14.7585,Z 58,A -151.0359,B 24.8343,C -2.9693,E1 24.8705,E2 -846.2271} C_DIS
LIN {X -20.4066,Y -13.2687,Z 58,A -155.2013,B 24.833,C -2.9806,E1 24.8641,E2 -842.0679} C_DIS
LIN {X -21.574,Y -11.2711,Z 58,A -161.0396,B 24.8317,C -2.9928,E1 24.8562,E2 -836.2282} C_DIS
LIN {X -22.4144,Y -9.4903,Z 58,A -165.0156,B 24.8298,C -3.0089,E1 24.8516,E2 -832.2689} C_DIS
LIN {X -22.9511,Y -8.1065,Z 58,A -168.6987,B 24.8288,C -3.0179,E1 24.8481,E2 -828.5865} C_DIS
LIN {X -23.3261,Y -6.9544,Z 58,A -171.5128,B 24.8278,C -3.0264,E1 24.8458,E2 -825.7766} C_DIS
LIN {X -23.7267,Y -5.4324,Z 58,A -175.4886,B 24.8267,C -3.0361,E1 24.8431,E2 -821.8007} C_DIS
LIN {X -24.0932,Y -3.4622,Z 58,A -179.679,B 24.8248,C -3.0529,E1 24.8412,E2 -817.6259} C_DIS
LIN {X -24.2238,Y -2.3844,Z 58,A 177.3636,B 24.8241,C -3.0589,E1 24.8403,E2 -814.6649} C_DIS
LIN {X -24.3327,Y -0.6295,Z 58,A 173.3373,B 24.8226,C -3.0722,E1 24.8398,E2 -810.6464} C_DIS
LIN {X -24.3175,Y 1.063,Z 58,A 168.774,B 24.8214,C -3.0819,E1 24.8401,E2 -806.0788} C_DIS
LIN {X -24.0948,Y 3.4483,Z 58,A 163.6367,B 24.8191,C -3.1019,E1 24.8418,E2 -800.9586} C_DIS
LIN {X -23.6713,Y 5.6685,Z 58,A 157.2123,B 24.8178,C -3.1131,E1 24.8455,E2 -794.5232} C_DIS
LIN {X -22.9825,Y 8.0172,Z 58,A 152.1546,B 24.8153,C -3.1338,E1 24.8499,E2 -789.4862} C_DIS
LIN {X -22.3303,Y 9.6865,Z 58,A 148.2351,B 24.8137,C -3.1477,E1 24.854,E2 -785.5783} C_DIS
LIN {X -21.6567,Y 11.111,Z 58,A 144.2805,B 24.8126,C -3.1572,E1 24.8589,E2 -781.625} C_DIS
LIN {X -21.0264,Y 12.2627,Z 58,A 141.0262,B 24.8116,C -3.165,E1 24.8634,E2 -778.3725} C_DIS
LIN {X -20.1861,Y 13.6004,Z 58,A 137.7275,B 24.8102,C -3.1773,E1 24.8684,E2 -775.0865} C_DIS
LIN {X -19.3964,Y 14.7057,Z 58,A 134.6163,B 24.8091,C -3.1861,E1 24.8735,E2 -771.9814} C_DIS
LIN {X -18.7193,Y 15.5581,Z 58,A 131.8919,B 24.8084,C -3.1918,E1 24.8783,E2 -769.2578} C_DIS
LIN {X -17.8107,Y 16.591,Z 58,A 128.5798,B 24.8075,C -3.1992,E1 24.8845,E2 -765.9489} C_DIS
LIN {X -16.7881,Y 17.6252,Z 58,A 124.8078,B 24.8068,C -3.2052,E1 24.8921,E2 -762.1755} C_DIS
LIN {X -15.6246,Y 18.6641,Z 58,A 121.6141,B 24.8055,C -3.2159,E1 24.8988,E2 -758.995} C_DIS
LIN {X -14.6549,Y 19.4346,Z 58,A 118.5619,B 24.8049,C -3.2212,E1 24.9055,E2 -755.9441} C_DIS
LIN {X -13.6317,Y 20.1655,Z 58,A 115.739,B 24.8041,C -3.2277,E1 24.912,E2 -753.1272} C_DIS
LIN {X -12.5356,Y 20.8646,Z 58,A 112.5398,B 24.8035,C -3.2324,E1 24.9196,E2 -749.9291} C_DIS
LIN {X -11.0412,Y 21.6924,Z 58,A 107.923,B 24.8031,C -3.2353,E1 24.931,E2 -745.3064} C_DIS
LIN {X -9.3951,Y 22.4545,Z 58,A 104.0411,B 24.8021,C -3.2438,E1 24.9409,E2 -741.4357} C_DIS
LIN {X -7.7885,Y 23.061,Z 58,A 100.0069,B 24.8015,C -3.2488,E1 24.9515,E2 -737.4055} C_DIS
LIN {X -6.2487,Y 23.5251,Z 58,A 96.1831,B 24.801,C -3.2525,E1 24.9617,E2 -733.5844} C_DIS
LIN {X -4.8146,Y 23.8599,Z 58,A 92.8415,B 24.8005,C -3.2563,E1 24.9708,E2 -730.2476} C_DIS
LIN {X -3.6113,Y 24.0715,Z 58,A 90.1719,B 24.8001,C -3.2598,E1 24.9782,E2 -727.5839} C_DIS
LIN {X -2.2423,Y 24.2372,Z 58,A 86.561,B 24.8002,C -3.2588,E1 24.9882,E2 -723.9685} C_DIS
LIN {X -0.7453,Y 24.3293,Z 58,A 83.2932,B 24.7999,C -3.262,E1 24.9973,E2 -720.7075} C_DIS
LIN {X 1.2132,Y 24.3103,Z 58,A 77.5648,B 24.8009,C -3.2538,E1 25.0134,E2 -714.9609} C_DIS
LIN {X 4.3336,Y 23.9518,Z 58,A 70.5637,B 24.8007,C -3.2551,E1 25.0327,E2 -707.9691} C_DIS
LIN {X 6.1683,Y 23.5464,Z 58,A 66.7469,B 24.8004,C -3.2577,E1 25.043,E2 -704.1642} C_DIS
LIN {X 7.544,Y 23.1421,Z 58,A 63.3556,B 24.8007,C -3.2551,E1 25.052,E2 -700.7727} C_DIS
LIN {X 8.8636,Y 22.6695,Z 58,A 60.1146,B 24.801,C -3.2526,E1 25.0605,E2 -697.5327} C_DIS
LIN {X 10.4006,Y 22.007,Z 58,A 55.8409,B 24.8019,C -3.2453,E1 25.0714,E2 -693.2522} C_DIS
LIN {X 12.4386,Y 20.9226,Z 58,A 50.0609,B 24.8032,C -3.2348,E1 25.0855,E2 -687.4643} C_DIS
LIN {X 14.005,Y 19.9081,Z 58,A 46.4273,B 24.8032,C -3.235,E1 25.0939,E2 -683.8435} C_DIS
LIN {X 15.2185,Y 18.9967,Z 58,A 42.7652,B 24.804,C -3.2279,E1 25.102,E2 -680.1779} C_DIS
LIN {X 16.309,Y 18.0692,Z 58,A 39.5361,B 24.8046,C -3.2228,E1 25.1087,E2 -676.9496} C_DIS
LIN {X 17.2649,Y 17.1578,Z 58,A 36.5711,B 24.8052,C -3.218,E1 25.1147,E2 -673.9854} C_DIS
LIN {X 18.0338,Y 16.3484,Z 58,A 33.8871,B 24.806,C -3.2117,E1 25.1198,E2 -671.2984} C_DIS
LIN {X 18.7168,Y 15.5612,Z 58,A 30.3398,B 24.808,C -3.1951,E1 25.1261,E2 -667.728} C_DIS
LIN {X 20.6084,Y 12.9525,Z 58,A 23.9515,B 24.8088,C -3.1889,E1 25.1363,E2 -661.3564} C_DIS
LIN {X 21.5301,Y 11.3545,Z 58,A 18.8812,B 24.811,C -3.1699,E1 25.1432,E2 -656.2673} C_DIS
Enddeposition()
END
